C07282=1082.479,167.330,-71.848,174.857,22.621,153.777
C07283=1082.484,167.580,-71.870,174.859,22.623,153.777
C07284=1082.490,167.828,-71.891,174.861,22.624,153.777
C07285=1082.495,168.078,-71.914,174.863,22.627,153.777
C07286=1082.500,168.327,-71.936,174.866,22.629,153.777
C07287=1082.506,168.576,-71.957,174.868,22.631,153.777
C07288=1082.511,168.825,-71.979,174.870,22.633,153.777
C07289=1082.517,169.074,-72.001,174.873,22.635,153.777
C07290=1082.522,169.323,-72.023,174.874,22.637,153.778
C07291=1082.528,169.572,-72.044,174.877,22.639,153.778
C07292=1082.533,169.820,-72.067,174.879,22.641,153.778
C07293=1082.539,170.069,-72.088,174.881,22.643,153.778
C07294=1082.544,170.318,-72.110,174.884,22.645,153.778
C07295=1082.550,170.567,-72.132,174.886,22.647,153.778
C07296=1082.556,170.817,-72.154,174.889,22.649,153.778
C07297=1082.561,171.066,-72.176,174.890,22.651,153.778
C07298=1082.567,171.315,-72.198,174.892,22.653,153.778
C07299=1082.572,171.563,-72.220,174.895,22.655,153.778
C07300=1082.578,171.812,-72.242,174.897,22.657,153.778
C07301=1082.583,172.062,-72.264,174.900,22.659,153.778
C07302=1082.589,172.310,-72.285,174.902,22.661,153.779
C07303=1082.595,172.559,-72.308,174.904,22.663,153.779
C07304=1082.599,172.808,-72.330,174.906,22.665,153.779
C07305=1082.606,173.057,-72.352,174.908,22.667,153.779
C07306=1082.611,173.307,-72.374,174.911,22.669,153.779
C07307=1082.617,173.555,-72.396,174.913,22.671,153.779
C07308=1082.622,173.804,-72.418,174.915,22.673,153.779
C07309=1082.628,174.054,-72.440,174.918,22.675,153.779
C07310=1082.634,174.302,-72.462,174.920,22.677,153.779
C07311=1082.639,174.551,-72.485,174.923,22.679,153.779
C07312=1082.645,174.800,-72.506,174.924,22.681,153.779
C07313=1082.650,175.049,-72.529,174.927,22.683,153.779
C07314=1082.657,175.328,-72.553,174.930,22.685,153.780
C07315=1082.663,175.607,-72.579,174.932,22.688,153.780
C07316=1082.669,175.887,-72.603,174.935,22.689,153.780
C07317=1082.676,176.166,-72.628,174.937,22.692,153.780
C07318=1082.681,176.415,-72.650,174.939,22.693,153.780
C07319=1082.686,176.664,-72.672,174.942,22.696,153.780
C07320=1082.693,176.913,-72.695,174.944,22.697,153.780
C07321=1082.698,177.162,-72.717,174.946,22.700,153.780
C07322=1082.703,177.410,-72.740,174.949,22.702,153.780
C07323=1082.709,177.660,-72.761,174.951,22.704,153.780
C07324=1082.715,177.909,-72.784,174.954,22.706,153.780
C07325=1082.721,178.158,-72.806,174.955,22.708,153.781
C07326=1082.726,178.406,-72.828,174.958,22.709,153.781
C07327=1082.732,178.655,-72.851,174.960,22.711,153.781
C07328=1082.738,178.904,-72.874,174.962,22.713,153.781
C07329=1082.744,179.154,-72.895,174.965,22.715,153.781
C07330=1082.749,179.402,-72.918,174.967,22.717,153.781
C07331=1082.754,179.651,-72.940,174.970,22.719,153.781
C07332=1082.761,179.900,-72.962,174.972,22.722,153.781
C07333=1082.766,180.149,-72.985,174.975,22.723,153.781
C07334=1082.772,180.398,-73.008,174.977,22.725,153.781
C07335=1082.777,180.646,-73.030,174.979,22.727,153.781
C07336=1082.783,180.896,-73.052,174.982,22.729,153.781
C07337=1082.789,181.145,-73.075,174.983,22.730,153.781
C07338=1082.794,181.394,-73.097,174.986,22.733,153.781
C07339=1082.801,181.643,-73.119,174.988,22.735,153.781
C07340=1082.806,181.891,-73.142,174.991,22.737,153.782
C07341=1082.811,182.140,-73.164,174.993,22.739,153.782
C07342=1082.817,182.389,-73.187,174.996,22.740,153.782
C07343=1082.824,182.638,-73.209,174.998,22.743,153.782
C07344=1082.829,182.887,-73.232,175.000,22.744,153.782
C07345=1082.835,183.136,-73.255,175.003,22.746,153.782
C07346=1082.841,183.385,-73.278,175.005,22.749,153.782
C07347=1082.846,183.634,-73.299,175.008,22.750,153.782
C07348=1082.852,183.883,-73.322,175.010,22.752,153.782
C07349=1082.858,184.131,-73.345,175.012,22.754,153.782
C07350=1082.863,184.380,-73.368,175.015,22.756,153.782
C07351=1082.869,184.630,-73.390,175.017,22.758,153.782
C07352=1082.875,184.878,-73.412,175.020,22.760,153.782
C07353=1082.881,185.127,-73.435,175.022,22.762,153.782
C07354=1082.887,185.376,-73.458,175.025,22.764,153.782
C07355=1082.891,185.625,-73.480,175.026,22.766,153.782
C07356=1082.896,185.874,-73.504,175.028,22.768,153.783
C07357=1082.902,186.123,-73.526,175.031,22.770,153.783
C07358=1082.908,186.372,-73.549,175.033,22.772,153.783
C07359=1082.913,186.620,-73.572,175.036,22.774,153.783
C07360=1082.919,186.869,-73.595,175.038,22.776,153.783
C07361=1082.924,187.119,-73.617,175.040,22.778,153.783
C07362=1082.930,187.368,-73.640,175.043,22.780,153.783
C07363=1082.935,187.617,-73.664,175.045,22.782,153.783
C07364=1082.940,187.865,-73.686,175.048,22.784,153.783
C07365=1082.946,188.114,-73.709,175.050,22.786,153.783
C07366=1082.951,188.363,-73.732,175.052,22.788,153.783
C07367=1082.957,188.612,-73.755,175.055,22.791,153.784
C07368=1082.963,188.861,-73.778,175.057,22.792,153.784
C07369=1082.968,189.110,-73.802,175.060,22.795,153.784
C07370=1082.974,189.359,-73.825,175.062,22.796,153.784
C07371=1082.979,189.607,-73.847,175.064,22.799,153.784
C07372=1082.985,189.856,-73.870,175.067,22.800,153.784
C07373=1082.990,190.105,-73.893,175.069,22.803,153.784
C07374=1082.995,190.354,-73.917,175.072,22.804,153.784
C07375=1083.001,190.603,-73.939,175.074,22.807,153.784
C07376=1083.007,190.852,-73.962,175.076,22.809,153.784
C07377=1083.012,191.101,-73.985,175.079,22.811,153.784
C07378=1083.018,191.379,-74.011,175.082,22.814,153.785
C07379=1083.024,191.658,-74.037,175.084,22.815,153.785
C07380=1083.031,191.937,-74.063,175.087,22.818,153.785
C07381=1083.037,192.217,-74.089,175.090,22.820,153.785
C07382=1083.042,192.466,-74.112,175.092,22.822,153.785
C07383=1083.049,192.714,-74.135,175.095,22.824,153.785
C07384=1083.054,192.962,-74.158,175.097,22.826,153.785
C07385=1083.059,193.211,-74.181,175.100,22.828,153.785
C07386=1083.064,193.460,-74.204,175.102,22.830,153.785
C07387=1083.070,193.709,-74.227,175.105,22.832,153.785
C07388=1083.076,193.958,-74.250,175.107,22.834,153.785
C07389=1083.081,194.207,-74.274,175.109,22.836,153.785
C07390=1083.087,194.456,-74.298,175.112,22.838,153.785
C07391=1083.093,194.704,-74.320,175.114,22.840,153.785
C07392=1083.098,194.954,-74.344,175.117,22.842,153.786
C07393=1083.103,195.203,-74.367,175.119,22.844,153.786
C07394=1083.109,195.451,-74.391,175.122,22.846,153.786
C07395=1083.115,195.700,-74.414,175.124,22.848,153.786
C07396=1083.120,195.949,-74.437,175.126,22.850,153.786
C07397=1083.126,196.198,-74.460,175.129,22.852,153.786
C07398=1083.132,196.446,-74.484,175.131,22.854,153.786
C07399=1083.137,196.695,-74.507,175.133,22.856,153.786
C07400=1083.143,196.944,-74.530,175.136,22.858,153.786
C07401=1083.149,197.194,-74.554,175.138,22.860,153.786
C07402=1083.154,197.442,-74.578,175.141,22.862,153.786
C07403=1083.160,197.691,-74.601,175.143,22.864,153.786
C07404=1083.166,197.940,-74.624,175.146,22.867,153.786
C07405=1083.171,198.189,-74.648,175.149,22.868,153.786
C07406=1083.177,198.438,-74.671,175.151,22.870,153.786
C07407=1083.183,198.686,-74.695,175.154,22.872,153.787
C07408=1083.188,198.935,-74.718,175.156,22.874,153.787
C07409=1083.193,199.184,-74.741,175.159,22.876,153.787
C07410=1083.200,199.432,-74.765,175.161,22.878,153.787
C07411=1083.204,199.682,-74.788,175.164,22.880,153.787
C07412=1083.211,199.931,-74.812,175.166,22.882,153.787
C07413=1083.217,200.179,-74.835,175.168,22.884,153.787
C07414=1083.222,200.429,-74.859,175.171,22.886,153.787
C07415=1083.228,200.677,-74.882,175.173,22.888,153.787
C07416=1083.234,200.926,-74.905,175.176,22.890,153.787
C07417=1083.239,201.174,-74.930,175.179,22.892,153.787
C07418=1083.245,201.423,-74.953,175.181,22.894,153.787
C07419=1083.251,201.673,-74.977,175.184,22.896,153.787
C07420=1083.256,201.921,-75.000,175.186,22.898,153.787
C07421=1083.262,202.170,-75.024,175.189,22.900,153.788
C07422=1083.267,202.419,-75.047,175.191,22.902,153.788
C07423=1083.273,202.667,-75.071,175.194,22.904,153.788
C07424=1083.279,202.916,-75.095,175.196,22.906,153.788
C07425=1083.285,203.165,-75.119,175.199,22.908,153.788
C07426=1083.290,203.414,-75.143,175.201,22.910,153.788
C07427=1083.295,203.663,-75.166,175.204,22.912,153.788
C07428=1083.301,203.911,-75.190,175.207,22.914,153.788
C07429=1083.307,204.160,-75.214,175.209,22.916,153.788
C07430=1083.312,204.409,-75.237,175.211,22.918,153.788
C07431=1083.318,204.658,-75.261,175.214,22.920,153.788
C07432=1083.323,204.907,-75.285,175.216,22.923,153.788
C07433=1083.329,205.156,-75.309,175.219,22.924,153.788
C07434=1083.335,205.404,-75.333,175.221,22.927,153.789
C07435=1083.340,205.653,-75.358,175.224,22.928,153.789
C07436=1083.346,205.902,-75.380,175.227,22.931,153.789
C07437=1083.351,206.150,-75.405,175.229,22.933,153.789
C07438=1083.357,206.400,-75.429,175.232,22.935,153.789
C07439=1083.363,206.649,-75.452,175.234,22.937,153.789
C07440=1083.368,206.897,-75.477,175.237,22.939,153.789
C07441=1083.373,207.146,-75.501,175.239,22.941,153.789
C07442=1083.397,208.176,-75.600,175.328,22.988,153.786
C07443=1083.406,208.569,-75.639,175.332,22.993,153.787
C07444=1083.415,208.961,-75.677,175.336,22.997,153.787
C07445=1083.423,209.353,-75.716,175.340,23.002,153.788
C07446=1083.432,209.746,-75.754,175.344,23.007,153.788
C07447=1083.438,209.995,-75.779,175.346,23.010,153.789
C07448=1083.444,210.243,-75.804,175.349,23.013,153.789
C07449=1083.450,210.492,-75.828,175.351,23.016,153.789
C07450=1083.455,210.741,-75.853,175.353,23.019,153.789
C07451=1083.460,210.990,-75.877,175.356,23.022,153.790
C07452=1083.466,211.238,-75.902,175.358,23.025,153.790
C07453=1083.472,211.487,-75.927,175.360,23.027,153.790
C07454=1083.478,211.736,-75.951,175.363,23.031,153.791
C07455=1083.483,211.984,-75.976,175.365,23.034,153.791
C07456=1083.489,212.233,-76.001,175.368,23.037,153.791
C07457=1083.494,212.482,-76.025,175.371,23.040,153.791
C07458=1083.501,212.731,-76.050,175.373,23.043,153.792
C07459=1083.506,212.979,-76.075,175.375,23.045,153.792
C07460=1083.512,213.229,-76.099,175.378,23.049,153.792
C07461=1083.517,213.476,-76.124,175.380,23.051,153.793
C07462=1083.523,213.726,-76.149,175.382,23.055,153.793
C07463=1083.528,213.975,-76.174,175.385,23.058,153.793
C07464=1083.534,214.223,-76.199,175.387,23.061,153.793
C07465=1083.539,214.472,-76.223,175.389,23.063,153.794
C07466=1083.546,214.721,-76.249,175.392,23.067,153.794
C07467=1083.551,214.969,-76.273,175.394,23.070,153.794
C07468=1083.557,215.218,-76.298,175.397,23.073,153.795
C07469=1083.562,215.467,-76.323,175.400,23.076,153.795
C07470=1083.568,215.715,-76.348,175.402,23.079,153.795
C07471=1083.573,215.964,-76.373,175.405,23.082,153.796
C07472=1083.579,216.213,-76.398,175.407,23.085,153.796
C07473=1083.585,216.461,-76.422,175.409,23.088,153.796
C07474=1083.590,216.710,-76.448,175.412,23.091,153.796
C07475=1083.596,216.959,-76.472,175.414,23.094,153.797
C07476=1083.602,217.208,-76.498,175.417,23.097,153.797
C07477=1083.607,217.456,-76.522,175.419,23.100,153.797
C07478=1083.612,217.705,-76.548,175.421,23.103,153.798
C07479=1083.619,217.954,-76.573,175.425,23.106,153.798
C07480=1083.624,218.202,-76.598,175.427,23.108,153.798
C07481=1083.630,218.451,-76.623,175.429,23.112,153.799
C07482=1083.636,218.699,-76.648,175.432,23.115,153.799
C07483=1083.641,218.949,-76.673,175.434,23.118,153.799
C07484=1083.647,219.197,-76.698,175.437,23.121,153.799
C07485=1083.653,219.445,-76.723,175.439,23.124,153.800
C07486=1083.658,219.695,-76.749,175.441,23.126,153.800
C07487=1083.664,219.943,-76.774,175.444,23.130,153.800
C07488=1083.670,220.191,-76.799,175.446,23.132,153.800
C07489=1083.676,220.441,-76.824,175.449,23.136,153.801
C07490=1083.681,220.689,-76.849,175.451,23.139,153.801
C07491=1083.687,220.938,-76.874,175.454,23.142,153.801
C07492=1083.693,221.186,-76.900,175.457,23.145,153.802
C07493=1083.697,221.435,-76.925,175.459,23.148,153.802
C07494=1083.704,221.684,-76.950,175.462,23.151,153.802
C07495=1083.713,222.080,-76.990,175.465,23.155,153.803
C07496=1083.722,222.477,-77.031,175.470,23.160,153.803
C07497=1083.730,222.873,-77.072,175.474,23.165,153.804
C07498=1083.740,223.270,-77.112,175.477,23.170,153.804
C07499=1083.745,223.518,-77.138,175.480,23.173,153.804
C07500=1083.751,223.767,-77.163,175.482,23.176,153.805
C07501=1083.757,224.016,-77.189,175.485,23.179,153.805
C07502=1083.762,224.264,-77.213,175.487,23.182,153.805
C07503=1083.768,224.513,-77.239,175.491,23.185,153.806
C07504=1083.774,224.762,-77.264,175.493,23.188,153.806
C07505=1083.779,225.010,-77.290,175.495,23.191,153.806
C07506=1083.785,225.259,-77.315,175.498,23.194,153.807
C07507=1083.790,225.508,-77.341,175.500,23.197,153.807
C07508=1083.797,225.757,-77.366,175.503,23.200,153.807
C07509=1083.801,226.005,-77.392,175.505,23.203,153.807
C07510=1083.807,226.254,-77.418,175.508,23.206,153.808
C07511=1083.813,226.502,-77.443,175.510,23.209,153.808
C07512=1083.819,226.751,-77.469,175.512,23.212,153.808
C07513=1083.824,226.999,-77.494,175.515,23.215,153.809
C07514=1083.830,227.248,-77.520,175.518,23.218,153.809
C07515=1083.836,227.496,-77.546,175.521,23.221,153.809
C07516=1083.842,227.745,-77.572,175.523,23.224,153.809
C07517=1083.847,227.993,-77.597,175.526,23.227,153.810
C07518=1083.853,228.242,-77.623,175.528,23.230,153.810
C07519=1083.858,228.491,-77.649,175.530,23.233,153.810
C07520=1083.864,228.740,-77.674,175.533,23.236,153.811
C07521=1083.870,228.989,-77.700,175.535,23.239,153.811
C07522=1083.875,229.237,-77.725,175.538,23.242,153.811
C07523=1083.881,229.485,-77.752,175.540,23.245,153.812
C07524=1083.887,229.734,-77.778,175.543,23.248,153.812
C07525=1083.893,229.983,-77.803,175.546,23.251,153.812
C07526=1083.898,230.232,-77.829,175.549,23.254,153.812
C07527=1083.904,230.480,-77.856,175.551,23.257,153.813
C07528=1083.910,230.728,-77.881,175.554,23.260,153.813
C07529=1083.915,230.977,-77.907,175.556,23.264,153.813
C07530=1083.921,231.226,-77.933,175.559,23.267,153.814
C07531=1083.926,231.475,-77.959,175.561,23.269,153.814
C07532=1083.933,231.723,-77.985,175.563,23.272,153.814
C07533=1083.938,231.972,-78.010,175.566,23.275,153.814
C07534=1083.943,232.220,-78.037,175.568,23.279,153.815
C07535=1083.949,232.469,-78.063,175.571,23.282,153.815
C07536=1083.955,232.718,-78.088,175.574,23.285,153.815
C07537=1083.961,232.966,-78.115,175.577,23.288,153.816
C07538=1083.966,233.215,-78.141,175.579,23.291,153.816
C07539=1083.972,233.464,-78.167,175.582,23.294,153.816
C07540=1083.977,233.712,-78.193,175.584,23.297,153.817
C07541=1083.983,233.961,-78.219,175.587,23.300,153.817
C07542=1083.989,234.209,-78.245,175.589,23.303,153.817
C07543=1083.994,234.458,-78.271,175.592,23.306,153.817
C07544=1084.000,234.706,-78.297,175.594,23.309,153.818
C07545=1084.005,234.955,-78.323,175.597,23.312,153.818
C07546=1084.011,235.204,-78.349,175.599,23.315,153.818
C07547=1084.020,235.591,-78.390,175.604,23.320,153.819
C07548=1084.029,235.979,-78.432,175.608,23.325,153.819
C07549=1084.037,236.367,-78.472,175.612,23.330,153.820
C07550=1084.047,236.755,-78.513,175.616,23.334,153.820
C07551=1084.052,237.004,-78.539,175.619,23.338,153.821
C07552=1084.058,237.253,-78.566,175.621,23.340,153.821
C07553=1084.063,237.500,-78.592,175.624,23.344,153.821
C07554=1084.069,237.749,-78.618,175.626,23.347,153.821
C07555=1084.075,237.998,-78.645,175.629,23.350,153.822
C07556=1084.080,238.247,-78.671,175.631,23.353,153.822
C07557=1084.086,238.495,-78.697,175.634,23.356,153.822
C07558=1084.092,238.743,-78.724,175.637,23.359,153.823
C07559=1084.097,238.992,-78.750,175.639,23.362,153.823
C07560=1084.103,239.241,-78.777,175.642,23.365,153.823
C07561=1084.109,239.489,-78.803,175.645,23.368,153.824
C07562=1084.114,239.737,-78.830,175.647,23.371,153.824
C07563=1084.120,239.986,-78.856,175.650,23.374,153.824
C07564=1084.126,240.235,-78.883,175.652,23.377,153.825
C07565=1084.132,240.484,-78.910,175.655,23.380,153.825
C07566=1084.138,240.732,-78.936,175.657,23.383,153.825
C07567=1084.143,240.981,-78.962,175.660,23.386,153.825
C07568=1084.149,241.230,-78.989,175.662,23.389,153.826
C07569=1084.155,241.478,-79.015,175.666,23.392,153.826
C07570=1084.160,241.727,-79.043,175.668,23.395,153.826
C07571=1084.166,241.975,-79.069,175.671,23.399,153.827
C07572=1084.171,242.224,-79.095,175.674,23.402,153.827
C07573=1084.177,242.472,-79.122,175.676,23.405,153.827
C07574=1084.183,242.721,-79.149,175.679,23.408,153.827
C07575=1084.188,242.969,-79.175,175.681,23.410,153.828
C07576=1084.194,243.217,-79.202,175.684,23.414,153.828
C07577=1084.200,243.466,-79.229,175.686,23.417,153.828
C07578=1084.205,243.714,-79.256,175.689,23.420,153.829
C07579=1084.211,243.963,-79.282,175.691,23.423,153.829
C07580=1084.217,244.212,-79.309,175.694,23.426,153.829
C07581=1084.223,244.460,-79.336,175.697,23.429,153.830
C07582=1084.228,244.709,-79.363,175.700,23.432,153.830
C07583=1084.234,244.957,-79.390,175.703,23.436,153.830
C07584=1084.239,245.206,-79.417,175.705,23.439,153.831
C07585=1084.244,245.454,-79.444,175.708,23.442,153.831
C07586=1084.250,245.703,-79.471,175.710,23.445,153.831
C07587=1084.256,245.951,-79.497,175.713,23.448,153.832
C07588=1084.262,246.199,-79.524,175.715,23.451,153.832
C07589=1084.267,246.449,-79.551,175.718,23.454,153.832
C07590=1084.273,246.697,-79.578,175.721,23.457,153.832
C07591=1084.279,246.945,-79.605,175.723,23.460,153.833
C07592=1084.284,247.194,-79.632,175.726,23.464,153.833
C07593=1084.290,247.442,-79.659,175.729,23.466,153.833
C07594=1084.295,247.690,-79.687,175.731,23.470,153.834
C07595=1084.301,247.939,-79.713,175.734,23.473,153.834
C07596=1084.307,248.187,-79.740,175.737,23.476,153.834
C07597=1084.312,248.437,-79.768,175.740,23.480,153.835
C07598=1084.318,248.685,-79.794,175.742,23.482,153.835
C07599=1084.326,249.066,-79.835,175.746,23.487,153.835
C07600=1084.335,249.447,-79.878,175.750,23.492,153.836
C07601=1084.343,249.828,-79.920,175.755,23.497,153.836
C07602=1084.351,250.209,-79.961,175.758,23.502,153.837
C07603=1084.357,250.457,-79.988,175.761,23.505,153.837
C07604=1084.363,250.706,-80.016,175.763,23.508,153.838
C07605=1084.369,250.955,-80.043,175.766,23.511,153.838
C07606=1084.374,251.203,-80.071,175.769,23.515,153.838
C07607=1084.380,251.451,-80.097,175.771,23.517,153.838
C07608=1084.385,251.700,-80.124,175.774,23.521,153.839
C07609=1084.392,251.948,-80.152,175.777,23.524,153.839
C07610=1084.397,252.197,-80.179,175.780,23.527,153.839
C07611=1084.402,252.445,-80.207,175.783,23.530,153.840
C07612=1084.408,252.693,-80.234,175.785,23.533,153.840
C07613=1084.413,252.943,-80.262,175.788,23.536,153.840
C07614=1084.419,253.190,-80.289,175.790,23.540,153.841
C07615=1084.424,253.439,-80.316,175.793,23.543,153.841
C07616=1084.431,253.687,-80.344,175.796,23.546,153.841
C07617=1084.436,253.936,-80.371,175.798,23.549,153.842
C07618=1084.442,254.184,-80.399,175.801,23.552,153.842
C07619=1084.447,254.433,-80.426,175.803,23.555,153.842
C07620=1084.453,254.681,-80.454,175.806,23.559,153.843
C07621=1084.459,254.930,-80.481,175.809,23.562,153.843
C07622=1084.464,255.178,-80.509,175.812,23.564,153.843
C07623=1084.470,255.427,-80.536,175.815,23.568,153.844
C07624=1084.476,255.675,-80.564,175.818,23.571,153.844
C07625=1084.481,255.923,-80.592,175.820,23.574,153.844
C07626=1084.488,256.172,-80.619,175.823,23.577,153.845
C07627=1084.493,256.420,-80.647,175.825,23.580,153.845
C07628=1084.498,256.669,-80.674,175.828,23.583,153.845
C07629=1084.505,256.917,-80.702,175.831,23.587,153.845
C07630=1084.510,257.165,-80.730,175.833,23.590,153.846
C07631=1084.515,257.414,-80.757,175.836,23.593,153.846
C07632=1084.522,257.662,-80.785,175.839,23.596,153.846
C07633=1084.527,257.910,-80.812,175.841,23.599,153.847
C07634=1084.533,258.158,-80.840,175.844,23.602,153.847
C07635=1084.539,258.408,-80.867,175.848,23.606,153.847
C07636=1084.544,258.656,-80.895,175.850,23.608,153.848
C07637=1084.550,258.904,-80.924,175.853,23.612,153.848
C07638=1084.556,259.152,-80.951,175.856,23.615,153.848
C07639=1084.562,259.401,-80.979,175.858,23.618,153.849
C07640=1084.567,259.650,-81.007,175.861,23.621,153.849
C07641=1084.573,259.897,-81.034,175.863,23.624,153.849
C07642=1084.579,260.146,-81.062,175.866,23.627,153.850
C07643=1084.585,260.394,-81.090,175.869,23.630,153.850
C07644=1084.590,260.643,-81.118,175.871,23.634,153.850
C07645=1084.596,260.891,-81.145,175.874,23.637,153.851
C07646=1084.602,261.140,-81.174,175.878,23.640,153.851
C07647=1084.608,261.388,-81.202,175.880,23.643,153.851
C07648=1084.614,261.637,-81.230,175.883,23.646,153.852
C07649=1084.620,261.884,-81.257,175.886,23.649,153.852
C07650=1084.626,262.133,-81.286,175.888,23.652,153.852
C07651=1084.635,262.511,-81.328,175.892,23.657,153.853
C07652=1084.644,262.889,-81.371,175.897,23.662,153.853
C07653=1084.652,263.268,-81.413,175.901,23.667,153.854
C07654=1084.661,263.647,-81.456,175.905,23.671,153.854
C07655=1084.666,263.895,-81.484,175.908,23.675,153.854
C07656=1084.672,264.144,-81.512,175.910,23.678,153.855
C07657=1084.678,264.391,-81.540,175.914,23.681,153.855
C07658=1084.685,264.639,-81.569,175.916,23.685,153.855
C07659=1084.690,264.888,-81.597,175.919,23.687,153.856
C07660=1084.695,265.137,-81.625,175.922,23.691,153.856
C07661=1084.701,265.385,-81.653,175.925,23.694,153.856
C07662=1084.707,265.633,-81.682,175.927,23.697,153.857
C07663=1084.712,265.881,-81.710,175.930,23.700,153.857
C07664=1084.718,266.130,-81.738,175.933,23.703,153.857
C07665=1084.723,266.378,-81.766,175.935,23.707,153.858
C07666=1084.729,266.626,-81.795,175.938,23.710,153.858
C07667=1084.735,266.874,-81.823,175.941,23.713,153.858
C07668=1084.741,267.123,-81.851,175.944,23.717,153.859
C07669=1084.747,267.372,-81.880,175.946,23.720,153.859
C07670=1084.752,267.620,-81.908,175.949,23.723,153.859
C07671=1084.758,267.868,-81.937,175.952,23.726,153.860
C07672=1084.764,268.116,-81.965,175.954,23.729,153.860
C07673=1084.770,268.365,-81.993,175.958,23.732,153.860
C07674=1084.775,268.612,-82.022,175.960,23.736,153.861
C07675=1084.781,268.861,-82.050,175.964,23.739,153.861
C07676=1084.787,269.110,-82.078,175.966,23.742,153.861
C07677=1084.792,269.358,-82.108,175.969,23.745,153.862
C07678=1084.798,269.606,-82.136,175.972,23.749,153.862
C07679=1084.803,269.854,-82.164,175.974,23.752,153.862
C07680=1084.810,270.103,-82.193,175.977,23.755,153.863
C07681=1084.815,270.351,-82.221,175.980,23.758,153.863
C07682=1084.821,270.599,-82.249,175.983,23.762,153.863
C07683=1084.826,270.848,-82.279,175.985,23.765,153.864
C07684=1084.832,271.097,-82.307,175.988,23.768,153.864
C07685=1084.838,271.344,-82.336,175.991,23.772,153.864
C07686=1084.844,271.593,-82.364,175.993,23.775,153.865
C07687=1084.849,271.841,-82.394,175.996,23.778,153.865
C07688=1084.855,272.089,-82.422,175.999,23.781,153.866
C07689=1084.861,272.337,-82.451,176.002,23.785,153.866
C07690=1084.866,272.585,-82.479,176.004,23.788,153.866
C07691=1084.872,272.834,-82.508,176.008,23.791,153.867
C07692=1084.878,273.083,-82.537,176.010,23.795,153.867
C07693=1084.884,273.331,-82.566,176.014,23.798,153.867
C07694=1084.889,273.579,-82.594,176.016,23.801,153.868
C07695=1084.895,273.827,-82.623,176.019,23.804,153.868
C07696=1084.901,274.075,-82.652,176.022,23.808,153.868
C07697=1084.906,274.323,-82.680,176.025,23.811,153.869
C07698=1084.912,274.572,-82.710,176.027,23.814,153.869
C07699=1084.918,274.820,-82.739,176.030,23.818,153.869
C07700=1084.924,275.068,-82.767,176.033,23.821,153.870
C07701=1084.929,275.316,-82.797,176.036,23.824,153.870
C07702=1084.935,275.565,-82.826,176.038,23.827,153.870
C07703=1084.944,275.946,-82.870,176.043,23.832,153.871
C07704=1084.953,276.328,-82.914,176.047,23.837,153.871
C07705=1084.961,276.708,-82.959,176.052,23.843,153.872
C07706=1084.970,277.089,-83.003,176.056,23.848,153.873
C07707=1084.976,277.338,-83.033,176.058,23.851,153.873
C07708=1084.981,277.586,-83.062,176.061,23.854,153.873
C07709=1084.988,277.834,-83.091,176.064,23.857,153.874
C07710=1084.992,278.082,-83.120,176.067,23.861,153.874
C07711=1084.998,278.331,-83.149,176.069,23.864,153.874
C07712=1085.004,278.579,-83.178,176.072,23.867,153.875
C07713=1085.010,278.827,-83.207,176.075,23.871,153.875
C07714=1085.016,279.076,-83.237,176.078,23.874,153.875
C07715=1085.021,279.323,-83.266,176.081,23.878,153.876
C07716=1085.027,279.571,-83.295,176.084,23.881,153.876
C07717=1085.033,279.820,-83.324,176.087,23.884,153.877
C07718=1085.039,280.068,-83.354,176.090,23.888,153.877
C07719=1085.045,280.316,-83.383,176.093,23.891,153.877
C07720=1085.050,280.565,-83.413,176.096,23.894,153.878
C07721=1085.056,280.812,-83.441,176.098,23.898,153.878
C07722=1085.061,281.060,-83.471,176.101,23.901,153.878
C07723=1085.068,281.309,-83.500,176.104,23.904,153.879
C07724=1085.073,281.557,-83.530,176.107,23.908,153.879
C07725=1085.079,281.805,-83.559,176.110,23.911,153.880
C07726=1085.084,282.054,-83.589,176.112,23.915,153.880
C07727=1085.090,282.301,-83.618,176.115,23.918,153.880
C07728=1085.095,282.550,-83.647,176.118,23.921,153.881
C07729=1085.101,282.798,-83.677,176.121,23.925,153.881
C07730=1085.107,283.046,-83.706,176.124,23.928,153.881
C07731=1085.113,283.295,-83.736,176.126,23.931,153.882
C07732=1085.119,283.543,-83.766,176.129,23.935,153.882
C07733=1085.123,283.790,-83.795,176.132,23.938,153.883
C07734=1085.130,284.039,-83.824,176.135,23.942,153.883
C07735=1085.135,284.287,-83.854,176.138,23.945,153.883
C07736=1085.141,284.535,-83.884,176.141,23.949,153.884
C07737=1085.147,284.783,-83.913,176.143,23.952,153.884
C07738=1085.153,285.031,-83.943,176.146,23.955,153.885
C07739=1085.158,285.280,-83.973,176.149,23.959,153.885
C07740=1085.164,285.528,-84.002,176.152,23.962,153.885
C07741=1085.170,285.776,-84.033,176.155,23.966,153.886
C07742=1085.176,286.024,-84.062,176.158,23.969,153.886
C07743=1085.181,286.273,-84.091,176.160,23.972,153.886
C07744=1085.187,286.520,-84.122,176.163,23.976,153.887
C07745=1085.193,286.769,-84.151,176.166,23.979,153.887
C07746=1085.199,287.017,-84.180,176.169,23.983,153.888
C07747=1085.205,287.265,-84.211,176.172,23.986,153.888
C07748=1085.210,287.513,-84.240,176.175,23.989,153.888
C07749=1085.215,287.760,-84.270,176.177,23.993,153.889
C07750=1085.221,288.009,-84.300,176.180,23.996,153.889
C07751=1085.227,288.257,-84.329,176.183,24.000,153.889
C07752=1085.233,288.505,-84.359,176.186,24.003,153.890
C07753=1085.239,288.754,-84.389,176.189,24.006,153.890
C07754=1085.245,289.002,-84.420,176.192,24.010,153.891
C07755=1085.253,289.392,-84.466,176.197,24.015,153.891
C07756=1085.263,289.783,-84.513,176.201,24.021,153.892
C07757=1085.272,290.174,-84.561,176.206,24.026,153.892
C07758=1085.281,290.565,-84.608,176.210,24.032,153.893
C07759=1085.287,290.813,-84.638,176.213,24.035,153.893
C07760=1085.292,291.061,-84.668,176.216,24.039,153.894
C07761=1085.298,291.309,-84.698,176.219,24.042,153.894
C07762=1085.304,291.557,-84.729,176.222,24.046,153.895
C07763=1085.309,291.805,-84.758,176.225,24.049,153.895
C07764=1085.315,292.053,-84.789,176.227,24.053,153.895
C07765=1085.321,292.301,-84.819,176.230,24.056,153.896
C07766=1085.326,292.549,-84.849,176.233,24.060,153.896
C07767=1085.333,292.798,-84.879,176.236,24.063,153.897
C07768=1085.339,293.046,-84.910,176.239,24.067,153.897
C07769=1085.344,293.294,-84.939,176.242,24.071,153.897
C07770=1085.350,293.542,-84.970,176.245,24.074,153.898
C07771=1085.355,293.790,-85.001,176.248,24.078,153.898
C07772=1085.361,294.038,-85.031,176.251,24.081,153.899
C07773=1085.367,294.286,-85.061,176.253,24.084,153.899
C07774=1085.372,294.534,-85.091,176.256,24.088,153.900
C07775=1085.378,294.782,-85.121,176.259,24.092,153.900
C07776=1085.384,295.030,-85.152,176.262,24.095,153.900
C07777=1085.390,295.278,-85.182,176.265,24.099,153.901
C07778=1085.396,295.526,-85.213,176.268,24.102,153.901
C07779=1085.402,295.774,-85.243,176.271,24.106,153.902
C07780=1085.407,296.022,-85.274,176.274,24.109,153.902
C07781=1085.413,296.270,-85.304,176.277,24.113,153.902
C07782=1085.418,296.518,-85.334,176.280,24.117,153.903
C07783=1085.425,296.767,-85.365,176.283,24.120,153.903
C07784=1085.431,297.015,-85.395,176.286,24.124,153.904
C07785=1085.436,297.263,-85.426,176.288,24.127,153.904
C07786=1085.441,297.511,-85.456,176.291,24.130,153.905
C07787=1085.447,297.758,-85.487,176.294,24.134,153.905
C07788=1085.453,298.006,-85.517,176.297,24.138,153.905
C07789=1085.459,298.255,-85.548,176.300,24.141,153.906
C07790=1085.465,298.503,-85.579,176.303,24.145,153.906
C07791=1085.470,298.750,-85.610,176.306,24.149,153.907
C07792=1085.476,298.998,-85.641,176.309,24.152,153.907
C07793=1085.482,299.246,-85.671,176.312,24.156,153.908
C07794=1085.487,299.494,-85.702,176.315,24.160,153.908
C07795=1085.493,299.742,-85.732,176.318,24.164,153.908
C07796=1085.498,299.991,-85.764,176.321,24.167,153.909
C07797=1085.504,300.239,-85.794,176.324,24.171,153.909
C07798=1085.509,300.487,-85.825,176.326,24.175,153.910
C07799=1085.515,300.734,-85.856,176.329,24.178,153.910
C07800=1085.520,300.982,-85.887,176.332,24.182,153.911
C07801=1085.527,301.231,-85.918,176.335,24.185,153.911
C07802=1085.532,301.479,-85.949,176.338,24.190,153.912
C07803=1085.538,301.726,-85.980,176.341,24.193,153.912
C07804=1085.543,301.974,-86.011,176.343,24.196,153.912
C07805=1085.549,302.222,-86.041,176.346,24.200,153.913
C07806=1085.555,302.471,-86.072,176.349,24.204,153.913
C07807=1085.564,302.875,-86.123,176.354,24.210,153.914
C07808=1085.573,303.280,-86.173,176.359,24.216,153.915
C07809=1085.583,303.685,-86.224,176.364,24.222,153.916
C07810=1085.592,304.089,-86.275,176.368,24.228,153.916
C07811=1085.597,304.338,-86.306,176.371,24.232,153.917
C07812=1085.604,304.586,-86.337,176.374,24.236,153.917
C07813=1085.609,304.834,-86.369,176.377,24.239,153.918
C07814=1085.615,305.081,-86.399,176.380,24.243,153.918
C07815=1085.621,305.330,-86.431,176.383,24.247,153.919
C07816=1085.627,305.577,-86.461,176.386,24.250,153.919
C07817=1085.632,305.825,-86.493,176.389,24.254,153.919
C07818=1085.638,306.074,-86.524,176.392,24.258,153.920
C07819=1085.644,306.321,-86.555,176.395,24.261,153.920
C07820=1085.649,306.569,-86.586,176.398,24.265,153.921
C07821=1085.656,306.817,-86.618,176.401,24.269,153.921
C07822=1085.661,307.064,-86.649,176.405,24.273,153.922
C07823=1085.667,307.313,-86.681,176.407,24.277,153.922
C07824=1085.673,307.561,-86.712,176.410,24.281,153.923
C07825=1085.678,307.809,-86.743,176.413,24.284,153.923
C07826=1085.684,308.057,-86.775,176.416,24.288,153.924
C07827=1085.690,308.304,-86.806,176.419,24.292,153.924
C07828=1085.696,308.553,-86.837,176.422,24.295,153.925
C07829=1085.702,308.800,-86.868,176.425,24.299,153.925
C07830=1085.708,309.048,-86.900,176.428,24.303,153.925
C07831=1085.713,309.296,-86.931,176.431,24.307,153.926
C07832=1085.720,309.544,-86.963,176.434,24.310,153.926
C07833=1085.725,309.792,-86.994,176.437,24.315,153.927
C07834=1085.731,310.040,-87.026,176.440,24.318,153.927
C07835=1085.737,310.288,-87.057,176.443,24.322,153.928
C07836=1085.743,310.536,-87.089,176.446,24.326,153.928
C07837=1085.748,310.784,-87.120,176.449,24.329,153.929
C07838=1085.754,311.032,-87.152,176.452,24.333,153.929
C07839=1085.760,311.279,-87.183,176.455,24.337,153.930
C07840=1085.766,311.528,-87.215,176.457,24.341,153.930
C07841=1085.771,311.775,-87.246,176.460,24.344,153.931
C07842=1085.778,312.023,-87.278,176.463,24.348,153.931
C07843=1085.783,312.271,-87.309,176.466,24.352,153.932
C07844=1085.789,312.519,-87.341,176.469,24.355,153.932
C07845=1085.795,312.767,-87.373,176.472,24.360,153.933
C07846=1085.802,313.014,-87.405,176.475,24.363,153.933
C07847=1085.807,313.263,-87.437,176.478,24.367,153.934
C07848=1085.813,313.510,-87.468,176.481,24.371,153.934
C07849=1085.819,313.758,-87.500,176.485,24.375,153.934
C07850=1085.826,314.006,-87.532,176.488,24.379,153.935
C07851=1085.831,314.254,-87.563,176.491,24.383,153.935
C07852=1085.837,314.502,-87.595,176.494,24.386,153.936
C07853=1085.843,314.750,-87.627,176.497,24.390,153.936
C07854=1085.848,314.998,-87.659,176.500,24.394,153.937
C07855=1085.854,315.246,-87.691,176.502,24.398,153.937
C07856=1085.860,315.493,-87.723,176.505,24.402,153.938
C07857=1085.866,315.742,-87.755,176.508,24.406,153.938
C07858=1085.872,315.990,-87.787,176.511,24.410,153.939
C07859=1085.880,316.398,-87.840,176.516,24.417,153.940
C07860=1085.890,316.805,-87.893,176.521,24.423,153.941
C07861=1085.899,317.213,-87.945,176.526,24.429,153.942
C07862=1085.909,317.621,-87.998,176.531,24.436,153.942
C07863=1085.914,317.869,-88.030,176.534,24.440,153.943
C07864=1085.920,318.117,-88.063,176.536,24.444,153.944
C07865=1085.925,318.364,-88.095,176.539,24.448,153.944
C07866=1085.931,318.612,-88.127,176.542,24.452,153.945
C07867=1085.937,318.859,-88.159,176.546,24.457,153.945
C07868=1085.942,319.108,-88.192,176.549,24.461,153.946
C07869=1085.948,319.356,-88.224,176.552,24.464,153.946
C07870=1085.954,319.603,-88.256,176.555,24.468,153.947
C07871=1085.960,319.851,-88.288,176.558,24.472,153.947
C07872=1085.965,320.100,-88.321,176.560,24.476,153.948
C07873=1085.971,320.346,-88.353,176.563,24.480,153.948
C07874=1085.977,320.595,-88.385,176.566,24.484,153.949
C07875=1085.983,320.843,-88.417,176.569,24.488,153.949
C07876=1085.989,321.091,-88.451,176.573,24.493,153.950
C07877=1085.994,321.338,-88.482,176.576,24.497,153.950
C07878=1086.000,321.586,-88.515,176.579,24.501,153.951
C07879=1086.006,321.834,-88.547,176.581,24.505,153.952
C07880=1086.012,322.082,-88.580,176.584,24.509,153.952
C07881=1086.017,322.330,-88.612,176.587,24.513,153.953
C07882=1086.023,322.577,-88.645,176.590,24.517,153.953
C07883=1086.029,322.826,-88.677,176.593,24.521,153.954
C07884=1086.035,323.073,-88.710,176.597,24.525,153.954
C07885=1086.041,323.321,-88.743,176.600,24.529,153.955
C07886=1086.046,323.569,-88.775,176.602,24.534,153.956
C07887=1086.052,323.816,-88.808,176.605,24.538,153.956
C07888=1086.058,324.065,-88.840,176.608,24.542,153.957
C07889=1086.064,324.312,-88.873,176.611,24.546,153.957
C07890=1086.070,324.560,-88.906,176.615,24.550,153.958
C07891=1086.076,324.808,-88.938,176.618,24.554,153.958
C07892=1086.081,325.055,-88.971,176.621,24.558,153.959
C07893=1086.087,325.303,-89.004,176.623,24.562,153.959
C07894=1086.093,325.551,-89.036,176.626,24.566,153.960
C07895=1086.099,325.799,-89.069,176.629,24.570,153.960
C07896=1086.105,326.047,-89.102,176.633,24.575,153.961
C07897=1086.111,326.294,-89.134,176.636,24.579,153.962
C07898=1086.117,326.543,-89.167,176.639,24.583,153.962
C07899=1086.123,326.790,-89.200,176.642,24.587,153.963
C07900=1086.129,327.038,-89.233,176.644,24.591,153.963
C07901=1086.135,327.286,-89.266,176.647,24.595,153.964
C07902=1086.141,327.533,-89.298,176.651,24.600,153.964
C07903=1086.146,327.781,-89.332,176.654,24.604,153.965
C07904=1086.152,328.029,-89.364,176.657,24.608,153.966
C07905=1086.158,328.277,-89.397,176.660,24.612,153.966
C07906=1086.164,328.524,-89.430,176.662,24.616,153.967
C07907=1086.169,328.772,-89.463,176.666,24.621,153.967
C07908=1086.176,329.020,-89.496,176.669,24.625,153.968
C07909=1086.182,329.268,-89.529,176.672,24.629,153.968
C07910=1086.188,329.515,-89.562,176.675,24.633,153.969
C07911=1086.198,329.916,-89.616,176.680,24.640,153.970
C07912=1086.207,330.318,-89.669,176.685,24.646,153.971
C07913=1086.217,330.719,-89.723,176.690,24.654,153.972
C07914=1086.227,331.120,-89.776,176.695,24.661,153.973
C07915=1086.233,331.367,-89.810,176.698,24.665,153.973
C07916=1086.239,331.615,-89.843,176.701,24.669,153.974
C07917=1086.244,331.863,-89.876,176.704,24.673,153.975
C07918=1086.251,332.111,-89.909,176.707,24.678,153.975
C07919=1086.256,332.358,-89.942,176.710,24.682,153.976
C07920=1086.262,332.606,-89.975,176.713,24.686,153.976
C07921=1086.268,332.854,-90.009,176.716,24.690,153.977
C07922=1086.274,333.101,-90.042,176.720,24.695,153.978
C07923=1086.279,333.349,-90.075,176.722,24.699,153.978
C07924=1086.285,333.597,-90.109,176.725,24.704,153.979
C07925=1086.291,333.845,-90.142,176.728,24.708,153.979
C07926=1086.296,334.092,-90.176,176.732,24.713,153.980
C07927=1086.303,334.340,-90.209,176.735,24.717,153.981
C07928=1086.308,334.588,-90.242,176.737,24.721,153.981
C07929=1086.314,334.835,-90.276,176.740,24.726,153.982
C07930=1086.320,335.083,-90.310,176.744,24.730,153.983
C07931=1086.326,335.332,-90.343,176.747,24.734,153.983
C07932=1086.332,335.579,-90.377,176.750,24.739,153.984
C07933=1086.338,335.826,-90.410,176.753,24.744,153.985
C07934=1086.344,336.074,-90.444,176.756,24.748,153.985
C07935=1086.349,336.322,-90.478,176.759,24.752,153.986
C07936=1086.355,336.570,-90.511,176.762,24.757,153.987
C07937=1086.361,336.817,-90.545,176.765,24.761,153.987
C07938=1086.368,337.065,-90.578,176.768,24.765,153.988
C07939=1086.374,337.312,-90.612,176.771,24.770,153.988
C07940=1086.379,337.560,-90.645,176.775,24.775,153.989
C07941=1086.385,337.808,-90.679,176.777,24.779,153.990
C07942=1086.391,338.055,-90.713,176.780,24.784,153.990
C07943=1086.396,338.303,-90.747,176.784,24.788,153.991
C07944=1086.403,338.551,-90.781,176.787,24.792,153.992
C07945=1086.408,338.799,-90.815,176.790,24.797,153.992
C07946=1086.414,339.046,-90.849,176.793,24.802,153.993
C07947=1086.420,339.294,-90.882,176.796,24.806,153.994
C07948=1086.426,339.541,-90.916,176.799,24.811,153.994
C07949=1086.432,339.788,-90.950,176.802,24.815,153.995
C07950=1086.438,340.037,-90.984,176.805,24.820,153.996
C07951=1086.444,340.284,-91.018,176.808,24.824,153.996
C07952=1086.449,340.532,-91.052,176.812,24.829,153.997
C07953=1086.455,340.779,-91.086,176.814,24.834,153.998
C07954=1086.461,341.027,-91.120,176.817,24.838,153.998
C07955=1086.467,341.275,-91.154,176.821,24.844,153.999
C07956=1086.472,341.522,-91.188,176.824,24.848,154.000
C07957=1086.478,341.770,-91.222,176.826,24.852,154.001
C07958=1086.484,342.018,-91.256,176.830,24.857,154.001
C07959=1086.490,342.266,-91.290,176.833,24.862,154.002
C07960=1086.496,342.513,-91.324,176.836,24.866,154.003
C07961=1086.502,342.760,-91.358,176.839,24.871,154.003
C07962=1086.509,343.008,-91.393,176.842,24.875,154.004
C07963=1086.518,343.403,-91.447,176.847,24.883,154.005
C07964=1086.527,343.799,-91.502,176.852,24.890,154.006
C07965=1086.537,344.194,-91.557,176.857,24.898,154.007
C07966=1086.546,344.589,-91.611,176.862,24.906,154.008
C07967=1086.552,344.836,-91.646,176.865,24.910,154.009
C07968=1086.558,345.084,-91.680,176.868,24.915,154.010
C07969=1086.564,345.332,-91.714,176.871,24.920,154.011
C07970=1086.570,345.579,-91.748,176.875,24.925,154.011
C07971=1086.576,345.827,-91.783,176.877,24.930,154.012
C07972=1086.581,346.075,-91.817,176.880,24.934,154.013
C07973=1086.587,346.322,-91.851,176.884,24.939,154.014
C07974=1086.593,346.570,-91.886,176.886,24.944,154.014
C07975=1086.599,346.817,-91.920,176.890,24.949,154.015
C07976=1086.605,347.064,-91.955,176.893,24.953,154.016
C07977=1086.611,347.312,-91.990,176.896,24.959,154.017
C07978=1086.617,347.560,-92.024,176.899,24.963,154.017
C07979=1086.622,347.808,-92.059,176.902,24.968,154.018
C07980=1086.628,348.055,-92.094,176.906,24.973,154.019
C07981=1086.634,348.302,-92.128,176.908,24.978,154.020
C07982=1086.640,348.550,-92.163,176.912,24.983,154.020
C07983=1086.646,348.798,-92.197,176.915,24.988,154.021
C07984=1086.652,349.045,-92.233,176.918,24.993,154.022
C07985=1086.658,349.293,-92.267,176.921,24.997,154.022
C07986=1086.664,349.540,-92.301,176.924,25.002,154.023
C07987=1086.670,349.787,-92.337,176.927,25.007,154.024
C07988=1086.676,350.035,-92.371,176.930,25.012,154.025
C07989=1086.681,350.283,-92.406,176.933,25.017,154.026
C07990=1086.687,350.530,-92.441,176.936,25.022,154.026
C07991=1086.693,350.778,-92.476,176.940,25.027,154.027
C07992=1086.699,351.025,-92.510,176.943,25.032,154.028
C07993=1086.705,351.273,-92.545,176.946,25.037,154.029
C07994=1086.711,351.520,-92.580,176.949,25.042,154.029
C07995=1086.717,351.768,-92.615,176.952,25.047,154.030
C07996=1086.723,352.015,-92.650,176.955,25.052,154.031
C07997=1086.729,352.263,-92.685,176.959,25.057,154.032
C07998=1086.735,352.510,-92.720,176.961,25.062,154.033
C07999=1086.741,352.758,-92.755,176.965,25.067,154.033
C08000=1086.747,353.005,-92.790,176.968,25.072,154.034
C08001=1086.753,353.252,-92.825,176.971,25.077,154.035
C08002=1086.759,353.500,-92.860,176.974,25.082,154.036
C08003=1086.765,353.747,-92.895,176.978,25.088,154.037
C08004=1086.771,353.995,-92.931,176.980,25.092,154.037
C08005=1086.776,354.242,-92.965,176.984,25.098,154.038
C08006=1086.783,354.490,-93.001,176.986,25.103,154.039
C08007=1086.788,354.737,-93.036,176.990,25.108,154.040
C08008=1086.794,354.985,-93.071,176.993,25.113,154.041
C08009=1086.800,355.232,-93.106,176.996,25.118,154.041
C08010=1086.806,355.479,-93.141,176.999,25.123,154.042
C08011=1086.812,355.727,-93.177,177.002,25.129,154.043
C08012=1086.818,355.974,-93.213,177.005,25.134,154.044
C08013=1086.824,356.222,-93.247,177.009,25.139,154.045
C08014=1086.829,356.469,-93.282,177.011,25.144,154.046
C08015=1086.839,356.867,-93.340,177.017,25.153,154.047
C08016=1086.849,357.265,-93.396,177.022,25.161,154.048
C08017=1086.859,357.663,-93.453,177.026,25.169,154.050
C08018=1086.868,358.061,-93.510,177.031,25.177,154.051
C08019=1086.874,358.309,-93.546,177.035,25.183,154.052
C08020=1086.879,358.556,-93.582,177.038,25.188,154.053
C08021=1086.886,358.803,-93.617,177.041,25.193,154.054
C08022=1086.892,359.051,-93.652,177.045,25.199,154.054
C08023=1086.898,359.299,-93.688,177.047,25.204,154.055
C08024=1086.904,359.546,-93.724,177.051,25.210,154.056
C08025=1086.910,359.793,-93.759,177.053,25.214,154.057
C08026=1086.916,360.041,-93.795,177.057,25.220,154.058
C08027=1086.922,360.287,-93.830,177.061,25.225,154.059
C08028=1086.928,360.535,-93.866,177.063,25.231,154.060
C08029=1086.934,360.782,-93.902,177.067,25.237,154.061
C08030=1086.940,361.030,-93.938,177.069,25.241,154.061
C08031=1086.946,361.277,-93.973,177.073,25.247,154.062
C08032=1086.952,361.525,-94.009,177.076,25.253,154.063
C08033=1086.958,361.772,-94.045,177.079,25.258,154.064
C08034=1086.964,362.019,-94.081,177.082,25.264,154.065
C08035=1086.970,362.266,-94.116,177.085,25.269,154.066
C08036=1086.976,362.513,-94.153,177.089,25.274,154.067
C08037=1086.982,362.761,-94.188,177.092,25.280,154.068
C08038=1086.988,363.009,-94.224,177.095,25.285,154.069
C08039=1086.994,363.255,-94.260,177.098,25.291,154.070
C08040=1087.000,363.503,-94.296,177.101,25.296,154.070
C08041=1087.006,363.750,-94.332,177.104,25.302,154.071
C08042=1087.012,363.997,-94.368,177.108,25.308,154.072
C08043=1087.018,364.245,-94.404,177.110,25.313,154.073
C08044=1087.024,364.491,-94.440,177.114,25.318,154.074
C08045=1087.030,364.739,-94.476,177.117,25.324,154.075
C08046=1087.035,364.987,-94.513,177.120,25.329,154.076
C08047=1087.041,365.234,-94.549,177.123,25.335,154.077
C08048=1087.048,365.481,-94.585,177.127,25.341,154.078
C08049=1087.054,365.729,-94.621,177.130,25.346,154.079
C08050=1087.060,365.976,-94.657,177.133,25.352,154.080
C08051=1087.066,366.223,-94.692,177.136,25.358,154.081
C08052=1087.071,366.470,-94.730,177.139,25.363,154.082
C08053=1087.078,366.717,-94.766,177.142,25.369,154.083
C08054=1087.084,366.965,-94.802,177.146,25.375,154.084
C08055=1087.090,367.212,-94.838,177.148,25.381,154.085
C08056=1087.096,367.459,-94.875,177.152,25.386,154.086
C08057=1087.101,367.706,-94.911,177.155,25.392,154.087
C08058=1087.107,367.954,-94.947,177.158,25.398,154.088
C08059=1087.113,368.201,-94.984,177.161,25.404,154.088
C08060=1087.119,368.449,-95.020,177.165,25.410,154.090
C08061=1087.125,368.696,-95.056,177.167,25.415,154.090
C08062=1087.131,368.943,-95.093,177.171,25.421,154.092
C08063=1087.137,369.190,-95.130,177.174,25.427,154.092
C08064=1087.144,369.437,-95.166,177.177,25.433,154.094
C08065=1087.149,369.684,-95.203,177.180,25.438,154.094
C08066=1087.155,369.932,-95.239,177.184,25.445,154.096
C08067=1087.166,370.345,-95.300,177.189,25.454,154.097
C08068=1087.176,370.759,-95.362,177.195,25.464,154.099
C08069=1087.185,371.173,-95.423,177.200,25.474,154.101
C08070=1087.196,371.586,-95.484,177.204,25.483,154.102
C08071=1087.202,371.834,-95.521,177.208,25.490,154.103
C08072=1087.208,372.081,-95.558,177.211,25.496,154.104
C08073=1087.214,372.328,-95.594,177.215,25.502,154.105
C08074=1087.220,372.575,-95.631,177.217,25.507,154.106
C08075=1087.226,372.822,-95.668,177.221,25.513,154.107
C08076=1087.232,373.070,-95.705,177.224,25.520,154.108
C08077=1087.238,373.317,-95.741,177.227,25.526,154.110
C08078=1087.245,373.563,-95.778,177.230,25.532,154.111
C08079=1087.251,373.811,-95.815,177.233,25.538,154.112
C08080=1087.257,374.058,-95.852,177.237,25.544,154.113
C08081=1087.262,374.305,-95.889,177.240,25.550,154.114
C08082=1087.268,374.552,-95.926,177.243,25.556,154.115
C08083=1087.275,374.799,-95.963,177.246,25.562,154.116
C08084=1087.280,375.046,-96.000,177.249,25.568,154.117
C08085=1087.286,375.294,-96.037,177.253,25.575,154.118
C08086=1087.293,375.541,-96.075,177.256,25.581,154.119
C08087=1087.299,375.788,-96.112,177.259,25.587,154.120
C08088=1087.304,376.035,-96.149,177.262,25.593,154.121
C08089=1087.311,376.282,-96.186,177.265,25.599,154.123
C08090=1087.317,376.529,-96.223,177.269,25.606,154.124
C08091=1087.322,376.777,-96.260,177.272,25.612,154.125
C08092=1087.329,377.023,-96.297,177.275,25.618,154.126
C08093=1087.334,377.270,-96.334,177.278,25.624,154.127
C08094=1087.340,377.517,-96.372,177.281,25.631,154.128
C08095=1087.347,377.765,-96.409,177.285,25.637,154.129
C08096=1087.353,378.012,-96.446,177.288,25.643,154.130
C08097=1087.359,378.259,-96.483,177.291,25.650,154.131
C08098=1087.365,378.506,-96.521,177.295,25.656,154.133
C08099=1087.371,378.752,-96.558,177.297,25.662,154.134
C08100=1087.377,379.000,-96.595,177.300,25.669,154.135
C08101=1087.383,379.247,-96.634,177.304,25.675,154.136
C08102=1087.390,379.494,-96.670,177.307,25.681,154.137
C08103=1087.396,379.741,-96.708,177.310,25.688,154.138
C08104=1087.402,379.987,-96.746,177.314,25.695,154.140
C08105=1087.407,380.235,-96.783,177.317,25.701,154.141
C08106=1087.414,380.482,-96.821,177.320,25.707,154.142
C08107=1087.420,380.729,-96.858,177.323,25.714,154.143
C08108=1087.426,380.975,-96.896,177.326,25.720,154.144
C08109=1087.432,381.224,-96.933,177.330,25.727,154.145
C08110=1087.438,381.470,-96.971,177.333,25.733,154.147
C08111=1087.445,381.717,-97.008,177.336,25.739,154.148
C08112=1087.451,381.963,-97.046,177.340,25.746,154.149
C08113=1087.457,382.211,-97.084,177.343,25.753,154.150
C08114=1087.463,382.458,-97.121,177.346,25.759,154.151
C08115=1087.469,382.705,-97.159,177.349,25.766,154.152
C08116=1087.475,382.952,-97.197,177.352,25.773,154.154
C08117=1087.481,383.199,-97.234,177.355,25.779,154.155
C08118=1087.487,383.446,-97.272,177.359,25.786,154.156
C08119=1087.496,383.796,-97.326,177.363,25.795,154.158
C08120=1087.504,384.147,-97.381,177.368,25.805,154.160
C08121=1087.513,384.497,-97.434,177.372,25.815,154.161
C08122=1087.522,384.847,-97.487,177.377,25.824,154.163
C08123=1087.528,385.094,-97.526,177.380,25.831,154.164
C08124=1087.534,385.341,-97.564,177.383,25.838,154.166
C08125=1087.540,385.588,-97.602,177.387,25.845,154.167
C08126=1087.546,385.836,-97.640,177.390,25.852,154.168
C08127=1087.552,386.082,-97.678,177.393,25.858,154.169
C08128=1087.558,386.329,-97.716,177.396,25.865,154.171
C08129=1087.565,386.576,-97.755,177.400,25.872,154.172
C08130=1087.571,386.823,-97.792,177.403,25.879,154.173
C08131=1087.577,387.070,-97.831,177.406,25.886,154.175
C08132=1087.583,387.317,-97.868,177.409,25.893,154.176
C08133=1087.589,387.563,-97.907,177.413,25.900,154.177
C08134=1087.595,387.811,-97.946,177.416,25.907,154.178
C08135=1087.601,388.057,-97.983,177.419,25.914,154.180
C08136=1087.608,388.304,-98.022,177.422,25.921,154.181
C08137=1087.614,388.551,-98.060,177.426,25.928,154.182
C08138=1087.620,388.798,-98.099,177.429,25.935,154.184
C08139=1087.626,389.045,-98.136,177.432,25.942,154.185
C08140=1087.632,389.292,-98.175,177.435,25.949,154.186
C08141=1087.638,389.538,-98.214,177.439,25.956,154.188
C08142=1087.645,389.786,-98.252,177.442,25.963,154.189
C08143=1087.651,390.032,-98.290,177.445,25.970,154.190
C08144=1087.657,390.279,-98.328,177.448,25.977,154.192
C08145=1087.663,390.526,-98.367,177.451,25.985,154.193
C08146=1087.670,390.773,-98.406,177.455,25.992,154.194
C08147=1087.676,391.020,-98.444,177.458,25.999,154.196
C08148=1087.682,391.266,-98.483,177.462,26.006,154.197
C08149=1087.689,391.514,-98.521,177.465,26.013,154.198
C08150=1087.694,391.760,-98.560,177.469,26.021,154.200
C08151=1087.701,392.007,-98.599,177.472,26.028,154.201
C08152=1087.708,392.254,-98.637,177.475,26.035,154.202
C08153=1087.713,392.501,-98.676,177.478,26.043,154.204
C08154=1087.720,392.748,-98.715,177.481,26.050,154.205
C08155=1087.725,392.994,-98.754,177.484,26.057,154.207
C08156=1087.732,393.242,-98.792,177.488,26.065,154.208
C08157=1087.738,393.489,-98.832,177.491,26.072,154.210
C08158=1087.744,393.735,-98.870,177.494,26.079,154.211
C08159=1087.750,393.982,-98.909,177.497,26.086,154.212
C08160=1087.757,394.229,-98.948,177.501,26.094,154.214
C08161=1087.763,394.475,-98.987,177.504,26.102,154.215
C08162=1087.769,394.722,-99.026,177.508,26.109,154.217
C08163=1087.778,395.060,-99.079,177.512,26.119,154.219
C08164=1087.786,395.399,-99.133,177.517,26.130,154.221
C08165=1087.795,395.736,-99.187,177.521,26.140,154.223
C08166=1087.803,396.074,-99.240,177.525,26.151,154.225
C08167=1087.809,396.321,-99.279,177.529,26.158,154.226
C08168=1087.816,396.568,-99.318,177.532,26.166,154.228
C08169=1087.822,396.814,-99.357,177.535,26.173,154.229
C08170=1087.828,397.062,-99.397,177.539,26.182,154.231
C08171=1087.834,397.289,-99.433,177.541,26.188,154.232
C08172=1087.840,397.517,-99.469,177.544,26.196,154.233
C08173=1087.845,397.744,-99.505,177.548,26.203,154.235
C08174=1087.851,397.972,-99.541,177.551,26.210,154.236
C08175=1087.857,398.200,-99.578,177.553,26.217,154.238
C08176=1087.863,398.428,-99.614,177.556,26.224,154.239
C08177=1087.868,398.655,-99.650,177.560,26.232,154.240
C08178=1087.874,398.882,-99.686,177.563,26.239,154.242
C08179=1087.880,399.129,-99.726,177.566,26.247,154.243
C08180=1087.886,399.377,-99.765,177.569,26.255,154.245
C08181=1087.893,399.623,-99.805,177.572,26.263,154.246
C08182=1087.899,399.870,-99.844,177.576,26.271,154.248
C08183=1087.905,400.116,-99.884,177.579,26.279,154.250
C08184=1087.911,400.363,-99.924,177.582,26.287,154.251
C08185=1087.917,400.610,-99.963,177.586,26.295,154.253
C08186=1087.924,400.857,-100.003,177.590,26.303,154.254
C08187=1087.930,401.104,-100.043,177.593,26.311,154.256
C08188=1087.937,401.350,-100.082,177.596,26.319,154.257
C08189=1087.943,401.597,-100.122,177.599,26.327,154.259
C08190=1087.949,401.844,-100.162,177.603,26.335,154.261
C08191=1087.956,402.091,-100.201,177.606,26.343,154.262
C08192=1087.962,402.337,-100.241,177.609,26.352,154.264
C08193=1087.968,402.584,-100.281,177.613,26.360,154.266
C08194=1087.974,402.831,-100.321,177.616,26.368,154.267
C08195=1087.981,403.077,-100.361,177.619,26.376,154.269
C08196=1087.987,403.325,-100.400,177.623,26.384,154.270
C08197=1087.993,403.571,-100.441,177.626,26.393,154.272
C08198=1088.000,403.818,-100.481,177.629,26.401,154.274
C08199=1088.006,404.065,-100.520,177.633,26.409,154.275
C08200=1088.012,404.311,-100.560,177.636,26.418,154.277
C08201=1088.018,404.558,-100.600,177.639,26.426,154.279
C08202=1088.025,404.804,-100.641,177.643,26.435,154.280
C08203=1088.031,405.051,-100.680,177.646,26.443,154.282
C08204=1088.037,405.298,-100.720,177.649,26.451,154.284
C08205=1088.044,405.544,-100.760,177.653,26.460,154.286
C08206=1088.050,405.791,-100.800,177.656,26.469,154.287
C08207=1088.056,406.037,-100.841,177.659,26.477,154.289
C08208=1088.063,406.284,-100.881,177.663,26.486,154.291
C08209=1088.068,406.531,-100.921,177.666,26.494,154.293
C08210=1088.075,406.778,-100.962,177.670,26.503,154.294
C08211=1088.082,407.024,-101.002,177.673,26.511,154.296
C08212=1088.088,407.271,-101.042,177.677,26.521,154.298
C08213=1088.095,407.518,-101.082,177.680,26.529,154.299
C08214=1088.101,407.764,-101.123,177.683,26.538,154.301
C08215=1088.107,408.011,-101.163,177.687,26.546,154.303
C08216=1088.113,408.257,-101.203,177.690,26.555,154.305
C08217=1088.120,408.505,-101.244,177.694,26.564,154.307
C08218=1088.126,408.751,-101.285,177.697,26.573,154.308
C08219=1088.132,408.998,-101.325,177.701,26.582,154.310
C08220=1088.139,409.244,-101.366,177.703,26.591,154.312
C08221=1088.144,409.491,-101.406,177.707,26.600,154.314
C08222=1088.151,409.737,-101.447,177.710,26.609,154.316
C08223=1088.157,409.985,-101.488,177.714,26.618,154.317
C08224=1088.164,410.231,-101.529,177.717,26.627,154.319
C08225=1088.170,410.477,-101.569,177.721,26.636,154.321
C08226=1088.176,410.724,-101.609,177.724,26.645,154.323
C08227=1088.182,410.952,-101.648,177.727,26.653,154.325
C08228=1088.188,411.180,-101.686,177.731,26.662,154.326
C08229=1088.194,411.409,-101.723,177.734,26.670,154.328
C08230=1088.200,411.637,-101.761,177.737,26.679,154.330
C08231=1088.206,411.864,-101.798,177.740,26.687,154.332
C08232=1088.211,412.093,-101.836,177.743,26.696,154.333
C08233=1088.217,412.321,-101.874,177.746,26.704,154.335
C08234=1088.224,412.549,-101.912,177.750,26.713,154.337
C08235=1088.230,412.796,-101.952,177.753,26.722,154.339
C08236=1088.236,413.043,-101.994,177.757,26.731,154.341
C08237=1088.243,413.289,-102.034,177.760,26.741,154.343
C08238=1088.249,413.536,-102.076,177.764,26.750,154.345
C08239=1088.256,413.782,-102.117,177.768,26.759,154.346
C08240=1088.262,414.029,-102.158,177.771,26.769,154.348
C08241=1088.269,414.275,-102.199,177.774,26.778,154.350
C08242=1088.275,414.522,-102.241,177.778,26.788,154.352
C08243=1088.282,414.769,-102.281,177.781,26.797,154.354
C08244=1088.288,415.015,-102.323,177.785,26.807,154.356
C08245=1088.295,415.261,-102.363,177.789,26.816,154.358
C08246=1088.301,415.508,-102.405,177.792,26.826,154.360
C08247=1088.308,415.754,-102.446,177.796,26.835,154.362
C08248=1088.314,416.001,-102.488,177.799,26.845,154.364
C08249=1088.320,416.248,-102.529,177.802,26.855,154.366
C08250=1088.327,416.494,-102.570,177.806,26.865,154.368
C08251=1088.333,416.740,-102.611,177.810,26.874,154.370
C08252=1088.340,416.987,-102.653,177.814,26.884,154.372
C08253=1088.346,417.233,-102.695,177.816,26.894,154.374
C08254=1088.353,417.480,-102.736,177.820,26.904,154.376
C08255=1088.359,417.726,-102.778,177.824,26.914,154.378
C08256=1088.366,417.972,-102.820,177.828,26.924,154.380
C08257=1088.372,418.219,-102.861,177.831,26.933,154.383
C08258=1088.379,418.465,-102.903,177.834,26.943,154.385
C08259=1088.385,418.711,-102.944,177.838,26.953,154.387
C08260=1088.392,418.958,-102.986,177.842,26.963,154.389
C08261=1088.398,419.205,-103.027,177.846,26.974,154.391
C08262=1088.404,419.451,-103.070,177.849,26.984,154.393
C08263=1088.411,419.698,-103.112,177.852,26.994,154.395
C08264=1088.418,419.944,-103.152,177.856,27.004,154.397
C08265=1088.424,420.190,-103.195,177.860,27.015,154.400
C08266=1088.430,420.436,-103.236,177.864,27.024,154.402
C08267=1088.437,420.683,-103.278,177.867,27.035,154.404
C08268=1088.444,420.929,-103.321,177.871,27.045,154.406
C08269=1088.450,421.176,-103.362,177.874,27.055,154.408
C08270=1088.457,421.422,-103.405,177.878,27.065,154.410
C08271=1088.464,421.668,-103.446,177.881,27.076,154.412
C08272=1088.470,421.914,-103.488,177.885,27.086,154.415
C08273=1088.477,422.161,-103.530,177.889,27.097,154.417
C08274=1088.484,422.407,-103.573,177.893,27.107,154.419
C08275=1088.490,422.653,-103.614,177.896,27.118,154.421
C08276=1088.496,422.900,-103.657,177.900,27.129,154.424
C08277=1088.503,423.146,-103.699,177.904,27.139,154.426
C08278=1088.509,423.393,-103.742,177.907,27.150,154.428
C08279=1088.515,423.639,-103.784,177.911,27.161,154.430
C08280=1088.522,423.885,-103.826,177.915,27.171,154.433
C08281=1088.529,424.132,-103.868,177.919,27.182,154.435
C08282=1088.535,424.378,-103.910,177.922,27.193,154.437
C08283=1088.542,424.614,-103.951,177.925,27.203,154.439
C08284=1088.547,424.849,-103.992,177.929,27.213,154.442
C08285=1088.554,425.085,-104.032,177.933,27.224,154.444
C08286=1088.561,425.322,-104.073,177.936,27.235,154.446
C08287=1088.567,425.557,-104.114,177.939,27.245,154.448
C08288=1088.573,425.793,-104.154,177.943,27.255,154.451
C08289=1088.579,426.029,-104.195,177.947,27.266,154.453
C08290=1088.586,426.264,-104.236,177.951,27.276,154.455
C08291=1088.593,426.511,-104.279,177.954,27.288,154.458
C08292=1088.599,426.757,-104.322,177.958,27.299,154.460
C08293=1088.606,427.004,-104.365,177.961,27.310,154.462
C08294=1088.613,427.250,-104.407,177.965,27.321,154.465
C08295=1088.619,427.495,-104.449,177.969,27.332,154.467
C08296=1088.625,427.742,-104.492,177.972,27.343,154.470
C08297=1088.632,427.988,-104.535,177.976,27.355,154.472
C08298=1088.639,428.234,-104.578,177.980,27.366,154.474
C08299=1088.646,428.480,-104.621,177.984,27.378,154.477
C08300=1088.652,428.727,-104.664,177.988,27.389,154.479
C08301=1088.659,428.973,-104.706,177.992,27.400,154.482
C08302=1088.666,429.219,-104.750,177.995,27.412,154.484
C08303=1088.672,429.465,-104.793,177.999,27.423,154.487
C08304=1088.679,429.711,-104.836,178.003,27.435,154.489
C08305=1088.685,429.958,-104.879,178.007,27.447,154.492
C08306=1088.692,430.204,-104.922,178.011,27.458,154.494
C08307=1088.699,430.450,-104.966,178.014,27.470,154.497
C08308=1088.706,430.696,-105.009,178.018,27.481,154.499
C08309=1088.713,430.942,-105.051,178.022,27.493,154.502
C08310=1088.719,431.188,-105.095,178.026,27.505,154.505
C08311=1088.726,431.434,-105.138,178.030,27.517,154.507
C08312=1088.732,431.680,-105.182,178.033,27.529,154.510
C08313=1088.740,431.926,-105.225,178.037,27.541,154.512
C08314=1088.746,432.172,-105.268,178.041,27.553,154.515
C08315=1088.753,432.418,-105.311,178.045,27.565,154.518
C08316=1088.759,432.664,-105.355,178.049,27.577,154.520
C08317=1088.765,432.911,-105.398,178.052,27.589,154.523
C08318=1088.773,433.156,-105.441,178.057,27.601,154.526
C08319=1088.779,433.402,-105.485,178.060,27.613,154.528
C08320=1088.785,433.648,-105.529,178.064,27.626,154.531
C08321=1088.793,433.894,-105.573,178.069,27.638,154.534
C08322=1088.800,434.140,-105.617,178.072,27.650,154.536
C08323=1088.806,434.386,-105.660,178.076,27.662,154.539
C08324=1088.813,434.632,-105.704,178.080,27.675,154.542
C08325=1088.820,434.878,-105.748,178.084,27.687,154.545
C08326=1088.826,435.124,-105.791,178.087,27.700,154.547
C08327=1088.832,435.370,-105.835,178.092,27.713,154.550
C08328=1088.840,435.616,-105.879,178.095,27.725,154.553
C08329=1088.847,435.862,-105.923,178.099,27.737,154.556
C08330=1088.853,436.108,-105.967,178.103,27.750,154.558
C08331=1088.860,436.354,-106.011,178.107,27.763,154.561
C08332=1088.866,436.600,-106.055,178.111,27.776,154.564
C08333=1088.874,436.846,-106.099,178.115,27.788,154.567
C08334=1088.881,437.091,-106.143,178.119,27.801,154.570
C08335=1088.887,437.337,-106.187,178.123,27.814,154.573
C08336=1088.894,437.584,-106.231,178.127,27.827,154.576
C08337=1088.901,437.829,-106.276,178.131,27.840,154.578
C08338=1088.907,438.075,-106.320,178.135,27.853,154.581
C08339=1088.916,438.371,-106.372,178.140,27.868,154.585
C08340=1088.925,438.667,-106.426,178.145,27.884,154.588
C08341=1088.933,438.962,-106.479,178.150,27.900,154.592
C08342=1088.941,439.258,-106.533,178.155,27.916,154.595
C08343=1088.948,439.504,-106.577,178.158,27.930,154.598
C08344=1088.955,439.750,-106.622,178.163,27.943,154.601
C08345=1088.962,439.995,-106.666,178.166,27.956,154.604
C08346=1088.969,440.242,-106.710,178.171,27.970,154.607
C08347=1088.976,440.487,-106.755,178.174,27.983,154.610
C08348=1088.983,440.733,-106.800,178.179,27.996,154.613
C08349=1088.990,440.978,-106.844,178.183,28.010,154.617
C08350=1088.996,441.224,-106.888,178.186,28.024,154.620
C08351=1089.003,441.471,-106.933,178.191,28.038,154.623
C08352=1089.010,441.716,-106.978,178.194,28.051,154.626
C08353=1089.017,441.962,-107.023,178.199,28.065,154.629
C08354=1089.023,442.208,-107.068,178.203,28.079,154.632
C08355=1089.031,442.454,-107.113,178.207,28.092,154.635
C08356=1089.037,442.699,-107.157,178.211,28.107,154.638
C08357=1089.045,442.945,-107.202,178.216,28.120,154.641
C08358=1089.052,443.190,-107.247,178.219,28.134,154.645
C08359=1089.058,443.436,-107.293,178.224,28.149,154.648
C08360=1089.065,443.681,-107.338,178.228,28.163,154.651
C08361=1089.072,443.928,-107.383,178.232,28.177,154.654
C08362=1089.080,444.174,-107.428,178.236,28.191,154.657
C08363=1089.086,444.419,-107.473,178.240,28.206,154.661
C08364=1089.093,444.665,-107.518,178.245,28.220,154.664
C08365=1089.100,444.910,-107.563,178.248,28.234,154.667
C08366=1089.107,445.156,-107.608,178.252,28.248,154.671
C08367=1089.114,445.402,-107.654,178.255,28.263,154.674
C08368=1089.122,445.648,-107.699,178.259,28.277,154.677
C08369=1089.128,445.893,-107.745,178.262,28.292,154.681
C08370=1089.135,446.139,-107.790,178.265,28.306,154.684
C08371=1089.143,446.384,-107.835,178.268,28.320,154.687
C08372=1089.149,446.630,-107.881,178.271,28.334,154.691
C08373=1089.157,446.876,-107.926,178.272,28.348,154.694
C08374=1089.163,447.122,-107.972,178.275,28.363,154.698
C08375=1089.171,447.367,-108.017,178.277,28.377,154.701
C08376=1089.177,447.612,-108.063,178.279,28.391,154.704
C08377=1089.184,447.858,-108.108,178.280,28.405,154.708
C08378=1089.191,448.104,-108.154,178.282,28.419,154.711
C08379=1089.199,448.350,-108.200,178.283,28.434,154.715
C08380=1089.206,448.596,-108.246,178.284,28.448,154.718
C08381=1089.213,448.841,-108.291,178.286,28.462,154.722
C08382=1089.220,449.086,-108.337,178.286,28.476,154.725
C08383=1089.227,449.332,-108.383,178.287,28.490,154.729
C08384=1089.234,449.577,-108.428,178.287,28.504,154.732
C08385=1089.242,449.822,-108.474,178.288,28.518,154.736
C08386=1089.252,450.069,-108.518,178.289,28.531,154.739
C08387=1088.872,450.060,-108.710,178.247,28.724,154.792
C08388=1088.862,449.813,-108.665,178.246,28.711,154.789
C08389=1088.853,449.568,-108.620,178.246,28.698,154.785
C08390=1088.847,449.323,-108.574,178.245,28.684,154.782
C08391=1088.839,449.078,-108.528,178.244,28.670,154.778
C08392=1088.832,448.832,-108.482,178.244,28.655,154.775
C08393=1088.825,448.586,-108.437,178.242,28.641,154.771
C08394=1088.818,448.340,-108.391,178.241,28.627,154.768
C08395=1088.811,448.096,-108.345,178.239,28.613,154.764
C08396=1088.804,447.850,-108.299,178.238,28.599,154.761
C08397=1088.797,447.604,-108.254,178.236,28.584,154.757
C08398=1088.790,447.358,-108.208,178.234,28.570,154.754
C08399=1088.782,447.113,-108.162,178.232,28.556,154.750
C08400=1088.775,446.867,-108.117,178.229,28.541,154.747
C08401=1088.769,446.621,-108.072,178.228,28.527,154.744
C08402=1088.761,446.376,-108.026,178.225,28.513,154.740
C08403=1088.754,446.130,-107.980,178.221,28.499,154.737
C08404=1088.747,445.884,-107.935,178.219,28.484,154.733
C08405=1088.740,445.639,-107.889,178.215,28.470,154.730
C08406=1088.733,445.393,-107.844,178.212,28.455,154.727
C08407=1088.726,445.148,-107.798,178.208,28.441,154.723
C08408=1088.720,444.902,-107.753,178.204,28.427,154.720
C08409=1088.712,444.656,-107.708,178.200,28.413,154.717
C08410=1088.705,444.411,-107.663,178.196,28.398,154.713
C08411=1088.699,444.165,-107.617,178.192,28.384,154.710
C08412=1088.691,443.919,-107.572,178.187,28.369,154.707
C08413=1088.684,443.673,-107.527,178.184,28.356,154.704
C08414=1088.677,443.428,-107.482,178.179,28.341,154.701
C08415=1088.670,443.182,-107.437,178.175,28.327,154.697
C08416=1088.664,442.936,-107.392,178.170,28.313,154.694
C08417=1088.656,442.691,-107.347,178.167,28.299,154.691
C08418=1088.649,442.445,-107.302,178.162,28.285,154.688
C08419=1088.642,442.199,-107.257,178.158,28.271,154.685
C08420=1088.635,441.953,-107.211,178.154,28.257,154.681
C08421=1088.629,441.708,-107.167,178.149,28.243,154.678
C08422=1088.621,441.462,-107.122,178.146,28.229,154.675
C08423=1088.614,441.216,-107.077,178.141,28.216,154.672
C08424=1088.607,440.970,-107.032,178.137,28.202,154.669
C08425=1088.600,440.725,-106.988,178.133,28.188,154.666
C08426=1088.593,440.478,-106.944,178.128,28.175,154.663
C08427=1088.587,440.233,-106.899,178.125,28.162,154.660
C08428=1088.580,439.988,-106.855,178.120,28.148,154.657
C08429=1088.573,439.742,-106.810,178.117,28.135,154.654
C08430=1088.566,439.496,-106.766,178.112,28.121,154.651
C08431=1088.559,439.249,-106.721,178.109,28.108,154.648
C08432=1088.551,438.967,-106.670,178.103,28.093,154.645
C08433=1088.543,438.685,-106.619,178.099,28.078,154.641
C08434=1088.535,438.402,-106.568,178.094,28.062,154.638
C08435=1088.527,438.120,-106.517,178.090,28.048,154.634
C08436=1088.520,437.874,-106.473,178.085,28.034,154.632
C08437=1088.513,437.628,-106.428,178.081,28.022,154.629
C08438=1088.506,437.382,-106.384,178.077,28.008,154.626
C08439=1088.500,437.137,-106.340,178.073,27.996,154.623
C08440=1088.493,436.890,-106.296,178.070,27.983,154.620
C08441=1088.485,436.644,-106.252,178.065,27.970,154.617
C08442=1088.479,436.399,-106.208,178.061,27.957,154.614
C08443=1088.472,436.153,-106.164,178.057,27.944,154.612
C08444=1088.465,435.906,-106.120,178.053,27.932,154.609
C08445=1088.459,435.661,-106.075,178.050,27.919,154.606
C08446=1088.451,435.415,-106.032,178.045,27.907,154.603
C08447=1088.445,435.169,-105.988,178.041,27.894,154.600
C08448=1088.438,434.923,-105.944,178.037,27.881,154.598
C08449=1088.431,434.677,-105.900,178.033,27.869,154.595
C08450=1088.424,434.431,-105.857,178.029,27.856,154.592
C08451=1088.418,434.185,-105.813,178.025,27.844,154.589
C08452=1088.411,433.939,-105.769,178.021,27.832,154.587
C08453=1088.405,433.693,-105.725,178.017,27.819,154.584
C08454=1088.398,433.447,-105.682,178.014,27.807,154.581
C08455=1088.391,433.201,-105.638,178.009,27.795,154.579
C08456=1088.384,432.955,-105.594,178.005,27.783,154.576
C08457=1088.377,432.709,-105.551,178.002,27.770,154.573
C08458=1088.371,432.463,-105.507,177.997,27.758,154.570
C08459=1088.364,432.217,-105.464,177.994,27.746,154.568
C08460=1088.358,431.971,-105.420,177.990,27.734,154.565
C08461=1088.350,431.725,-105.377,177.986,27.722,154.563
C08462=1088.344,431.479,-105.333,177.982,27.710,154.560
C08463=1088.337,431.233,-105.291,177.978,27.699,154.557
C08464=1088.331,430.987,-105.247,177.974,27.686,154.555
C08465=1088.323,430.741,-105.203,177.971,27.675,154.552
C08466=1088.317,430.494,-105.160,177.967,27.663,154.550
C08467=1088.310,430.248,-105.117,177.962,27.651,154.547
C08468=1088.304,430.002,-105.074,177.958,27.640,154.545
C08469=1088.296,429.756,-105.031,177.955,27.628,154.542
C08470=1088.291,429.510,-104.988,177.951,27.616,154.539
C08471=1088.284,429.265,-104.944,177.947,27.605,154.537
C08472=1088.278,429.018,-104.901,177.944,27.593,154.534
C08473=1088.270,428.772,-104.858,177.940,27.582,154.532
C08474=1088.264,428.526,-104.816,177.935,27.570,154.530
C08475=1088.257,428.279,-104.772,177.932,27.558,154.527
C08476=1088.250,428.034,-104.729,177.928,27.547,154.525
C08477=1088.243,427.787,-104.687,177.924,27.536,154.522
C08478=1088.237,427.541,-104.644,177.920,27.525,154.520
C08479=1088.230,427.295,-104.601,177.917,27.514,154.517
C08480=1088.224,427.048,-104.558,177.913,27.502,154.515
C08481=1088.216,426.803,-104.515,177.909,27.491,154.512
C08482=1088.210,426.556,-104.473,177.905,27.480,154.510
C08483=1088.203,426.310,-104.430,177.902,27.469,154.508
C08484=1088.197,426.074,-104.389,177.898,27.458,154.505
C08485=1088.190,425.837,-104.348,177.894,27.448,154.503
C08486=1088.184,425.601,-104.308,177.890,27.437,154.501
C08487=1088.178,425.364,-104.266,177.886,27.426,154.499
C08488=1088.172,425.128,-104.226,177.883,27.416,154.496
C08489=1088.165,424.892,-104.185,177.880,27.406,154.494
C08490=1088.159,424.655,-104.144,177.876,27.395,154.492
C08491=1088.153,424.418,-104.103,177.872,27.384,154.490
C08492=1088.146,424.172,-104.061,177.868,27.373,154.487
C08493=1088.139,423.926,-104.018,177.865,27.363,154.485
C08494=1088.133,423.679,-103.976,177.862,27.352,154.483
C08495=1088.126,423.434,-103.934,177.858,27.342,154.480
C08496=1088.120,423.187,-103.892,177.854,27.331,154.478
C08497=1088.113,422.941,-103.849,177.850,27.320,154.476
C08498=1088.107,422.695,-103.807,177.847,27.309,154.474
C08499=1088.101,422.448,-103.765,177.843,27.299,154.471
C08500=1088.093,422.202,-103.723,177.839,27.289,154.469
C08501=1088.086,421.956,-103.680,177.835,27.278,154.467
C08502=1088.080,421.709,-103.639,177.831,27.267,154.465
C08503=1088.074,421.463,-103.596,177.828,27.257,154.463
C08504=1088.067,421.216,-103.554,177.824,27.246,154.460
C08505=1088.061,420.971,-103.512,177.821,27.236,154.458
C08506=1088.054,420.724,-103.470,177.817,27.226,154.456
C08507=1088.047,420.477,-103.428,177.813,27.216,154.454
C08508=1088.041,420.231,-103.386,177.809,27.205,154.452
C08509=1088.035,419.984,-103.344,177.806,27.195,154.449
C08510=1088.027,419.738,-103.302,177.802,27.185,154.447
C08511=1088.021,419.492,-103.261,177.799,27.175,154.445
C08512=1088.015,419.245,-103.219,177.795,27.165,154.443
C08513=1088.008,418.999,-103.177,177.791,27.155,154.441
C08514=1088.002,418.753,-103.135,177.787,27.145,154.439
C08515=1087.995,418.506,-103.094,177.783,27.135,154.437
C08516=1087.989,418.260,-103.053,177.781,27.124,154.435
C08517=1087.982,418.014,-103.010,177.777,27.114,154.433
C08518=1087.976,417.768,-102.969,177.773,27.104,154.430
C08519=1087.969,417.521,-102.927,177.769,27.094,154.428
C08520=1087.963,417.275,-102.886,177.766,27.085,154.426
C08521=1087.956,417.028,-102.844,177.762,27.075,154.424
C08522=1087.950,416.782,-102.803,177.759,27.065,154.422
C08523=1087.944,416.535,-102.761,177.755,27.055,154.420
C08524=1087.938,416.289,-102.719,177.752,27.046,154.418
C08525=1087.930,416.042,-102.678,177.748,27.036,154.416
C08526=1087.924,415.796,-102.637,177.744,27.026,154.414
C08527=1087.917,415.549,-102.595,177.741,27.016,154.412
C08528=1087.911,415.303,-102.554,177.737,27.007,154.410
C08529=1087.904,415.056,-102.513,177.733,26.997,154.408
C08530=1087.898,414.809,-102.472,177.730,26.988,154.406
C08531=1087.891,414.563,-102.431,177.726,26.978,154.404
C08532=1087.885,414.317,-102.389,177.723,26.968,154.402
C08533=1087.878,414.070,-102.348,177.720,26.959,154.400
C08534=1087.872,413.823,-102.307,177.716,26.950,154.398
C08535=1087.865,413.577,-102.266,177.712,26.940,154.396
C08536=1087.859,413.330,-102.225,177.709,26.931,154.394
C08537=1087.852,413.085,-102.184,177.705,26.921,154.393
C08538=1087.846,412.837,-102.143,177.702,26.912,154.391
C08539=1087.839,412.591,-102.102,177.698,26.903,154.389
C08540=1087.834,412.362,-102.064,177.695,26.894,154.387
C08541=1087.827,412.133,-102.025,177.692,26.885,154.385
C08542=1087.821,411.905,-101.988,177.688,26.877,154.383
C08543=1087.816,411.676,-101.950,177.685,26.869,154.382
C08544=1087.810,411.448,-101.912,177.682,26.860,154.380
C08545=1087.804,411.218,-101.874,177.678,26.852,154.378
C08546=1087.798,410.990,-101.836,177.675,26.843,154.376
C08547=1087.792,410.761,-101.799,177.672,26.834,154.375
C08548=1087.785,410.514,-101.757,177.668,26.825,154.373
C08549=1087.779,410.268,-101.717,177.665,26.817,154.371
C08550=1087.773,410.021,-101.676,177.661,26.807,154.369
C08551=1087.767,409.775,-101.635,177.658,26.798,154.367
C08552=1087.760,409.528,-101.595,177.654,26.789,154.365
C08553=1087.754,409.281,-101.554,177.651,26.780,154.364
C08554=1087.748,409.034,-101.514,177.647,26.771,154.362
C08555=1087.741,408.789,-101.473,177.644,26.762,154.360
C08556=1087.735,408.542,-101.432,177.640,26.753,154.358
C08557=1087.729,408.295,-101.392,177.637,26.744,154.356
C08558=1087.722,408.048,-101.352,177.633,26.736,154.355
C08559=1087.716,407.801,-101.311,177.630,26.727,154.353
C08560=1087.710,407.555,-101.270,177.627,26.718,154.351
C08561=1087.703,407.309,-101.230,177.623,26.709,154.349
C08562=1087.697,407.062,-101.190,177.620,26.701,154.347
C08563=1087.691,406.815,-101.149,177.616,26.692,154.346
C08564=1087.684,406.568,-101.108,177.613,26.683,154.344
C08565=1087.678,406.322,-101.068,177.610,26.675,154.342
C08566=1087.671,406.075,-101.028,177.606,26.666,154.340
C08567=1087.665,405.829,-100.988,177.603,26.657,154.339
C08568=1087.659,405.582,-100.948,177.599,26.649,154.337
C08569=1087.653,405.335,-100.908,177.596,26.640,154.335
C08570=1087.647,405.088,-100.868,177.593,26.632,154.334
C08571=1087.641,404.842,-100.827,177.589,26.623,154.332
C08572=1087.634,404.595,-100.787,177.586,26.615,154.330
C08573=1087.628,404.349,-100.747,177.583,26.607,154.329
C08574=1087.621,404.101,-100.707,177.579,26.598,154.327
C08575=1087.615,403.854,-100.667,177.576,26.590,154.325
C08576=1087.608,403.608,-100.627,177.573,26.581,154.324
C08577=1087.602,403.361,-100.587,177.569,26.573,154.322
C08578=1087.596,403.115,-100.547,177.566,26.565,154.320
C08579=1087.590,402.868,-100.507,177.563,26.556,154.319
C08580=1087.583,402.621,-100.467,177.558,26.548,154.317
C08581=1087.577,402.374,-100.428,177.555,26.540,154.315
C08582=1087.570,402.128,-100.388,177.552,26.532,154.314
C08583=1087.564,401.881,-100.348,177.549,26.523,154.312
C08584=1087.558,401.634,-100.309,177.545,26.515,154.311
C08585=1087.551,401.388,-100.268,177.542,26.507,154.309
C08586=1087.545,401.140,-100.229,177.539,26.499,154.307
C08587=1087.539,400.894,-100.189,177.536,26.491,154.306
C08588=1087.533,400.647,-100.150,177.532,26.483,154.304
C08589=1087.527,400.401,-100.110,177.529,26.474,154.302
C08590=1087.521,400.154,-100.070,177.526,26.467,154.301
C08591=1087.514,399.908,-100.031,177.522,26.459,154.299
C08592=1087.508,399.661,-99.991,177.518,26.450,154.298
C08593=1087.501,399.413,-99.952,177.515,26.442,154.296
C08594=1087.495,399.167,-99.912,177.512,26.435,154.295
C08595=1087.489,398.920,-99.872,177.509,26.427,154.293
C08596=1087.483,398.692,-99.836,177.506,26.420,154.292
C08597=1087.477,398.464,-99.800,177.502,26.412,154.290
C08598=1087.472,398.236,-99.763,177.499,26.405,154.289
C08599=1087.466,398.008,-99.727,177.497,26.398,154.287
C08600=1087.460,397.779,-99.691,177.493,26.391,154.286
C08601=1087.454,397.551,-99.654,177.490,26.383,154.285
C08602=1087.448,397.323,-99.618,177.487,26.376,154.283
C08603=1087.443,397.095,-99.582,177.484,26.369,154.282
C08604=1087.436,396.848,-99.543,177.480,26.361,154.280
C08605=1087.430,396.602,-99.503,177.477,26.354,154.279
C08606=1087.424,396.355,-99.464,177.474,26.346,154.277
C08607=1087.417,396.108,-99.425,177.471,26.338,154.276
C08608=1087.411,395.861,-99.385,177.468,26.331,154.274
C08609=1087.405,395.614,-99.347,177.465,26.323,154.273
C08610=1087.399,395.368,-99.307,177.461,26.315,154.271
C08611=1087.393,395.121,-99.268,177.457,26.308,154.270
C08612=1087.386,394.874,-99.229,177.454,26.300,154.268
C08613=1087.381,394.627,-99.190,177.451,26.293,154.267
C08614=1087.374,394.381,-99.151,177.448,26.285,154.266
C08615=1087.368,394.134,-99.112,177.444,26.277,154.264
C08616=1087.361,393.886,-99.074,177.441,26.270,154.263
C08617=1087.356,393.640,-99.035,177.438,26.263,154.261
C08618=1087.349,393.393,-98.996,177.435,26.255,154.260
C08619=1087.344,393.146,-98.957,177.431,26.248,154.258
C08620=1087.337,392.900,-98.918,177.428,26.240,154.257
C08621=1087.330,392.653,-98.879,177.425,26.233,154.255
C08622=1087.325,392.406,-98.841,177.421,26.225,154.254
C08623=1087.318,392.159,-98.802,177.418,26.218,154.253
C08624=1087.312,391.912,-98.762,177.414,26.211,154.251
C08625=1087.306,391.666,-98.724,177.411,26.204,154.250
C08626=1087.299,391.418,-98.686,177.408,26.196,154.249
C08627=1087.294,391.172,-98.647,177.405,26.189,154.247
C08628=1087.287,390.924,-98.609,177.401,26.182,154.246
C08629=1087.280,390.677,-98.570,177.398,26.175,154.244
C08630=1087.274,390.431,-98.531,177.395,26.168,154.243
C08631=1087.268,390.184,-98.493,177.392,26.160,154.242
C08632=1087.262,389.937,-98.454,177.388,26.153,154.240
C08633=1087.256,389.690,-98.416,177.385,26.146,154.239
C08634=1087.249,389.443,-98.377,177.382,26.139,154.238
C08635=1087.243,389.196,-98.339,177.379,26.132,154.236
C08636=1087.237,388.949,-98.300,177.375,26.125,154.235
C08637=1087.231,388.703,-98.262,177.372,26.117,154.234
C08638=1087.224,388.456,-98.223,177.369,26.110,154.232
C08639=1087.218,388.209,-98.186,177.366,26.103,154.231
C08640=1087.212,387.962,-98.147,177.362,26.096,154.230
C08641=1087.206,387.715,-98.109,177.359,26.089,154.228
C08642=1087.200,387.468,-98.071,177.356,26.082,154.227
C08643=1087.194,387.222,-98.032,177.352,26.075,154.226
C08644=1087.188,386.975,-97.994,177.349,26.069,154.225
C08645=1087.181,386.727,-97.956,177.346,26.062,154.223
C08646=1087.175,386.481,-97.918,177.342,26.055,154.222
C08647=1087.169,386.234,-97.879,177.339,26.048,154.221
C08648=1087.163,385.987,-97.842,177.336,26.041,154.219
C08649=1087.157,385.740,-97.804,177.333,26.034,154.218
C08650=1087.151,385.493,-97.765,177.329,26.027,154.217
C08651=1087.145,385.246,-97.727,177.326,26.020,154.216
C08652=1087.139,385.025,-97.693,177.323,26.014,154.214
C08653=1087.133,384.803,-97.659,177.320,26.008,154.213
C08654=1087.128,384.582,-97.625,177.317,26.002,154.212
C08655=1087.123,384.361,-97.591,177.314,25.995,154.211
C08656=1087.117,384.139,-97.557,177.311,25.990,154.210
C08657=1087.111,383.918,-97.523,177.309,25.984,154.209
C08658=1087.106,383.697,-97.489,177.306,25.977,154.208
C08659=1087.101,383.476,-97.455,177.303,25.972,154.207
C08660=1087.095,383.229,-97.417,177.300,25.965,154.205
C08661=1087.088,382.982,-97.379,177.296,25.958,154.204
C08662=1087.082,382.735,-97.341,177.293,25.951,154.203
C08663=1087.077,382.488,-97.303,177.290,25.944,154.202
C08664=1087.070,382.241,-97.266,177.286,25.938,154.200
C08665=1087.064,381.994,-97.228,177.283,25.931,154.199
C08666=1087.058,381.747,-97.191,177.280,25.925,154.198
C08667=1087.052,381.499,-97.153,177.277,25.918,154.197
C08668=1087.046,381.253,-97.115,177.274,25.912,154.196
C08669=1087.040,381.006,-97.077,177.270,25.905,154.194
C08670=1087.033,380.759,-97.040,177.267,25.899,154.193
C08671=1087.027,380.511,-97.003,177.264,25.892,154.192
C08672=1087.021,380.265,-96.965,177.260,25.886,154.191
C08673=1087.016,380.018,-96.927,177.257,25.879,154.190
C08674=1087.008,379.771,-96.890,177.254,25.873,154.189
C08675=1087.003,379.523,-96.853,177.251,25.867,154.188
C08676=1086.997,379.277,-96.815,177.248,25.860,154.186
C08677=1086.991,379.030,-96.777,177.244,25.854,154.185
C08678=1086.984,378.782,-96.740,177.241,25.847,154.184
C08679=1086.978,378.535,-96.702,177.238,25.841,154.183
C08680=1086.972,378.288,-96.665,177.235,25.834,154.182
C08681=1086.967,378.041,-96.628,177.232,25.828,154.181
C08682=1086.960,377.795,-96.591,177.228,25.822,154.179
C08683=1086.954,377.548,-96.553,177.225,25.816,154.178
C08684=1086.948,377.300,-96.515,177.222,25.809,154.177
C08685=1086.941,377.053,-96.479,177.218,25.803,154.176
C08686=1086.936,376.806,-96.441,177.216,25.797,154.175
C08687=1086.930,376.559,-96.404,177.212,25.791,154.174
C08688=1086.924,376.312,-96.367,177.209,25.784,154.173
C08689=1086.918,376.065,-96.330,177.205,25.778,154.172
C08690=1086.912,375.818,-96.293,177.202,25.771,154.170
C08691=1086.906,375.571,-96.255,177.200,25.765,154.169
C08692=1086.900,375.324,-96.219,177.196,25.759,154.168
C08693=1086.894,375.076,-96.181,177.193,25.753,154.167
C08694=1086.888,374.829,-96.144,177.189,25.747,154.166
C08695=1086.881,374.582,-96.107,177.187,25.741,154.165
C08696=1086.876,374.335,-96.070,177.184,25.734,154.164
C08697=1086.869,374.088,-96.034,177.180,25.728,154.163
C08698=1086.864,373.841,-95.996,177.177,25.722,154.162
C08699=1086.857,373.594,-95.959,177.174,25.716,154.161
C08700=1086.852,373.347,-95.922,177.171,25.710,154.160
C08701=1086.845,373.100,-95.886,177.167,25.704,154.159
C08702=1086.840,372.852,-95.849,177.164,25.698,154.158
C08703=1086.833,372.606,-95.812,177.161,25.692,154.156
C08704=1086.827,372.359,-95.775,177.158,25.686,154.155
C08705=1086.821,372.111,-95.738,177.154,25.680,154.154
C08706=1086.815,371.864,-95.702,177.151,25.674,154.153
C08707=1086.809,371.617,-95.665,177.148,25.668,154.152
C08708=1086.799,371.202,-95.603,177.143,25.658,154.151
C08709=1086.789,370.787,-95.541,177.137,25.648,154.149
C08710=1086.778,370.373,-95.480,177.132,25.638,154.147
C08711=1086.768,369.958,-95.418,177.127,25.628,154.145
C08712=1086.760,369.605,-95.367,177.122,25.620,154.144
C08713=1086.751,369.253,-95.314,177.118,25.612,154.143
C08714=1086.742,368.899,-95.262,177.113,25.603,154.141
C08715=1086.734,368.547,-95.210,177.108,25.595,154.140
C08716=1086.727,368.300,-95.174,177.105,25.589,154.139
C08717=1086.721,368.052,-95.138,177.102,25.583,154.138
C08718=1086.716,367.805,-95.101,177.099,25.577,154.137
C08719=1086.710,367.558,-95.065,177.096,25.572,154.136
C08720=1086.704,367.311,-95.028,177.092,25.566,154.135
C08721=1086.698,367.064,-94.993,177.089,25.560,154.134
C08722=1086.692,366.816,-94.956,177.086,25.555,154.133
C08723=1086.686,366.569,-94.919,177.083,25.548,154.132
C08724=1086.680,366.322,-94.883,177.080,25.543,154.131
C08725=1086.674,366.074,-94.846,177.077,25.537,154.130
C08726=1086.669,365.827,-94.811,177.073,25.531,154.129
C08727=1086.662,365.580,-94.775,177.070,25.525,154.128
C08728=1086.656,365.333,-94.738,177.067,25.520,154.127
C08729=1086.650,365.085,-94.702,177.064,25.514,154.126
C08730=1086.644,364.838,-94.666,177.060,25.509,154.125
C08731=1086.638,364.591,-94.630,177.058,25.503,154.124
C08732=1086.632,364.343,-94.593,177.054,25.498,154.123
C08733=1086.627,364.096,-94.558,177.052,25.492,154.122
C08734=1086.620,363.849,-94.521,177.048,25.487,154.121
C08735=1086.614,363.602,-94.486,177.044,25.481,154.120
C08736=1086.608,363.354,-94.450,177.042,25.476,154.119
C08737=1086.602,363.107,-94.413,177.038,25.470,154.119
C08738=1086.596,362.859,-94.378,177.035,25.464,154.118
C08739=1086.590,362.613,-94.342,177.032,25.459,154.117
C08740=1086.584,362.365,-94.306,177.029,25.453,154.116
C08741=1086.578,362.118,-94.270,177.026,25.448,154.115
C08742=1086.572,361.870,-94.235,177.023,25.442,154.114
C08743=1086.566,361.624,-94.198,177.019,25.437,154.113
C08744=1086.560,361.376,-94.163,177.016,25.432,154.112
C08745=1086.554,361.128,-94.127,177.013,25.426,154.111
C08746=1086.548,360.880,-94.091,177.010,25.420,154.110
C08747=1086.542,360.634,-94.055,177.007,25.415,154.109
C08748=1086.536,360.386,-94.019,177.004,25.410,154.109
C08749=1086.530,360.139,-93.984,177.000,25.404,154.108
C08750=1086.524,359.891,-93.949,176.997,25.398,154.107
C08751=1086.518,359.644,-93.913,176.994,25.394,154.106
C08752=1086.512,359.397,-93.877,176.991,25.388,154.105
C08753=1086.506,359.149,-93.842,176.988,25.383,154.104
C08754=1086.500,358.903,-93.806,176.984,25.377,154.103
C08755=1086.494,358.655,-93.770,176.982,25.372,154.102
C08756=1086.488,358.408,-93.735,176.978,25.367,154.101
C08757=1086.482,358.161,-93.699,176.976,25.362,154.101
C08758=1086.476,357.913,-93.664,176.972,25.356,154.100
C08759=1086.470,357.665,-93.628,176.968,25.351,154.099
C08760=1086.463,357.372,-93.586,176.965,25.345,154.098
C08761=1086.455,357.079,-93.545,176.962,25.338,154.097
C08762=1086.449,356.785,-93.502,176.957,25.332,154.096
C08763=1086.441,356.492,-93.461,176.954,25.326,154.095
C08764=1086.436,356.245,-93.425,176.950,25.320,154.094
C08765=1086.430,355.997,-93.390,176.948,25.316,154.093
C08766=1086.424,355.750,-93.355,176.944,25.310,154.092
C08767=1086.418,355.503,-93.319,176.941,25.305,154.092
C08768=1086.412,355.254,-93.284,176.938,25.300,154.091
C08769=1086.407,355.007,-93.249,176.935,25.295,154.090
C08770=1086.400,354.760,-93.214,176.932,25.290,154.089
C08771=1086.394,354.513,-93.178,176.929,25.285,154.088
C08772=1086.389,354.265,-93.143,176.925,25.279,154.087
C08773=1086.383,354.018,-93.108,176.923,25.274,154.087
C08774=1086.377,353.770,-93.073,176.919,25.269,154.086
C08775=1086.370,353.523,-93.037,176.916,25.264,154.085
C08776=1086.365,353.275,-93.003,176.913,25.259,154.084
C08777=1086.359,353.028,-92.967,176.910,25.254,154.083
C08778=1086.353,352.780,-92.932,176.906,25.248,154.083
C08779=1086.347,352.533,-92.897,176.904,25.244,154.082
C08780=1086.341,352.286,-92.862,176.900,25.238,154.081
C08781=1086.335,352.038,-92.828,176.897,25.233,154.080
C08782=1086.329,351.791,-92.792,176.895,25.229,154.079
C08783=1086.323,351.543,-92.758,176.891,25.223,154.078
C08784=1086.317,351.296,-92.722,176.888,25.218,154.078
C08785=1086.311,351.048,-92.688,176.885,25.213,154.077
C08786=1086.306,350.801,-92.653,176.882,25.208,154.076
C08787=1086.299,350.553,-92.618,176.878,25.203,154.075
C08788=1086.294,350.306,-92.583,176.876,25.199,154.075
C08789=1086.287,350.058,-92.548,176.872,25.193,154.074
C08790=1086.282,349.810,-92.514,176.869,25.188,154.073
C08791=1086.275,349.563,-92.479,176.866,25.183,154.072
C08792=1086.270,349.316,-92.445,176.863,25.178,154.071
C08793=1086.263,349.068,-92.409,176.860,25.174,154.071
C08794=1086.258,348.821,-92.375,176.857,25.169,154.070
C08795=1086.252,348.572,-92.340,176.854,25.164,154.069
C08796=1086.246,348.326,-92.305,176.850,25.159,154.068
C08797=1086.241,348.078,-92.270,176.847,25.154,154.068
C08798=1086.234,347.830,-92.236,176.845,25.149,154.067
C08799=1086.228,347.583,-92.202,176.841,25.144,154.066
C08800=1086.222,347.335,-92.166,176.838,25.139,154.065
C08801=1086.216,347.088,-92.132,176.835,25.134,154.065
C08802=1086.211,346.841,-92.098,176.832,25.130,154.064
C08803=1086.205,346.592,-92.063,176.828,25.124,154.063
C08804=1086.199,346.345,-92.029,176.825,25.120,154.062
C08805=1086.193,346.098,-91.995,176.823,25.115,154.062
C08806=1086.187,345.850,-91.959,176.819,25.110,154.061
C08807=1086.181,345.603,-91.925,176.816,25.105,154.060
C08808=1086.175,345.355,-91.891,176.813,25.100,154.059
C08809=1086.170,345.107,-91.856,176.810,25.096,154.059
C08810=1086.164,344.860,-91.822,176.807,25.091,154.058
C08811=1086.157,344.612,-91.788,176.804,25.086,154.057
C08812=1086.149,344.216,-91.733,176.799,25.078,154.056
C08813=1086.139,343.820,-91.678,176.794,25.071,154.055
C08814=1086.129,343.424,-91.623,176.789,25.063,154.054
C08815=1086.120,343.027,-91.568,176.784,25.056,154.053
C08816=1086.114,342.780,-91.534,176.781,25.051,154.052
C08817=1086.108,342.533,-91.500,176.778,25.047,154.051
C08818=1086.101,342.285,-91.466,176.774,25.042,154.051
C08819=1086.096,342.037,-91.432,176.772,25.037,154.050
C08820=1086.090,341.789,-91.398,176.769,25.032,154.049
C08821=1086.085,341.542,-91.364,176.765,25.028,154.048
C08822=1086.078,341.294,-91.329,176.762,25.023,154.048
C08823=1086.073,341.047,-91.295,176.760,25.019,154.047
C08824=1086.067,340.799,-91.261,176.756,25.014,154.046
C08825=1086.061,340.551,-91.228,176.753,25.009,154.046
C08826=1086.055,340.303,-91.193,176.750,25.004,154.045
C08827=1086.049,340.056,-91.159,176.747,25.000,154.044
C08828=1086.043,339.808,-91.126,176.744,24.995,154.044
C08829=1086.037,339.561,-91.092,176.741,24.991,154.043
C08830=1086.032,339.314,-91.058,176.737,24.986,154.042
C08831=1086.025,339.065,-91.024,176.735,24.982,154.042
C08832=1086.020,338.818,-90.990,176.732,24.977,154.041
C08833=1086.014,338.570,-90.956,176.728,24.972,154.040
C08834=1086.008,338.323,-90.923,176.725,24.968,154.040
C08835=1086.002,338.075,-90.889,176.722,24.963,154.039
C08836=1085.996,337.827,-90.855,176.720,24.959,154.038
C08837=1085.990,337.579,-90.821,176.716,24.954,154.038
C08838=1085.985,337.331,-90.788,176.713,24.950,154.037
C08839=1085.979,337.084,-90.754,176.710,24.945,154.036
C08840=1085.973,336.837,-90.720,176.707,24.940,154.036
C08841=1085.967,336.589,-90.687,176.704,24.936,154.035
C08842=1085.961,336.341,-90.653,176.701,24.932,154.034
C08843=1085.955,336.093,-90.619,176.697,24.927,154.034
C08844=1085.949,335.846,-90.586,176.694,24.923,154.033
C08845=1085.943,335.598,-90.552,176.692,24.918,154.032
C08846=1085.938,335.350,-90.518,176.689,24.914,154.032
C08847=1085.932,335.103,-90.484,176.685,24.909,154.031
C08848=1085.926,334.855,-90.452,176.682,24.905,154.030
C08849=1085.920,334.608,-90.418,176.679,24.901,154.030
C08850=1085.914,334.360,-90.384,176.677,24.896,154.029
C08851=1085.908,334.112,-90.350,176.673,24.891,154.028
C08852=1085.902,333.864,-90.317,176.670,24.887,154.028
C08853=1085.896,333.616,-90.284,176.667,24.883,154.027
C08854=1085.890,333.369,-90.250,176.664,24.878,154.026
C08855=1085.885,333.121,-90.217,176.661,24.874,154.026
C08856=1085.879,332.873,-90.184,176.658,24.870,154.025
C08857=1085.873,332.625,-90.151,176.655,24.865,154.025
C08858=1085.867,332.378,-90.117,176.652,24.861,154.024
C08859=1085.861,332.130,-90.084,176.648,24.856,154.023
C08860=1085.856,331.882,-90.050,176.646,24.852,154.023
C08861=1085.850,331.635,-90.017,176.643,24.847,154.022
C08862=1085.844,331.387,-89.984,176.640,24.843,154.021
C08863=1085.838,331.139,-89.951,176.637,24.839,154.021
C08864=1085.828,330.737,-89.897,176.632,24.832,154.020
C08865=1085.819,330.336,-89.843,176.627,24.825,154.019
C08866=1085.808,329.934,-89.790,176.622,24.818,154.018
C08867=1085.799,329.532,-89.736,176.617,24.812,154.017
C08868=1085.793,329.284,-89.704,176.614,24.807,154.016
C08869=1085.787,329.036,-89.670,176.611,24.803,154.016
C08870=1085.781,328.789,-89.638,176.608,24.799,154.015
C08871=1085.776,328.541,-89.604,176.604,24.794,154.015
C08872=1085.769,328.293,-89.571,176.601,24.790,154.014
C08873=1085.764,328.045,-89.538,176.598,24.786,154.014
C08874=1085.757,327.798,-89.505,176.596,24.782,154.013
C08875=1085.751,327.550,-89.473,176.593,24.778,154.012
C08876=1085.746,327.302,-89.440,176.589,24.774,154.012
C08877=1085.740,327.054,-89.407,176.586,24.769,154.011
C08878=1085.734,326.806,-89.374,176.583,24.765,154.011
C08879=1085.728,326.559,-89.341,176.580,24.761,154.010
C08880=1085.721,326.311,-89.308,176.577,24.757,154.010
C08881=1085.716,326.063,-89.275,176.575,24.753,154.009
C08882=1085.710,325.815,-89.243,176.571,24.748,154.008
C08883=1085.704,325.567,-89.210,176.568,24.744,154.008
C08884=1085.698,325.319,-89.177,176.565,24.740,154.007
C08885=1085.693,325.072,-89.145,176.562,24.736,154.007
C08886=1085.687,324.824,-89.112,176.559,24.732,154.006
C08887=1085.681,324.576,-89.079,176.556,24.728,154.005
C08888=1085.675,324.329,-89.047,176.554,24.724,154.005
C08889=1085.669,324.080,-89.014,176.550,24.719,154.004
C08890=1085.663,323.833,-88.981,176.547,24.715,154.004
C08891=1085.657,323.584,-88.949,176.544,24.711,154.003
C08892=1085.652,323.337,-88.916,176.541,24.707,154.003
C08893=1085.646,323.090,-88.883,176.538,24.703,154.002
C08894=1085.640,322.841,-88.851,176.535,24.699,154.002
C08895=1085.634,322.594,-88.818,176.532,24.695,154.001
C08896=1085.628,322.345,-88.786,176.529,24.690,154.000
C08897=1085.623,322.098,-88.754,176.526,24.686,154.000
C08898=1085.617,321.850,-88.721,176.523,24.682,153.999
C08899=1085.611,321.602,-88.688,176.520,24.678,153.999
C08900=1085.605,321.354,-88.656,176.517,24.674,153.998
C08901=1085.599,321.107,-88.624,176.514,24.670,153.998
C08902=1085.594,320.859,-88.591,176.511,24.666,153.997
C08903=1085.588,320.611,-88.559,176.508,24.662,153.997
C08904=1085.582,320.363,-88.526,176.506,24.658,153.996
C08905=1085.576,320.116,-88.494,176.502,24.654,153.995
C08906=1085.571,319.867,-88.461,176.499,24.649,153.995
C08907=1085.565,319.619,-88.429,176.496,24.645,153.994
C08908=1085.559,319.372,-88.397,176.493,24.641,153.994
C08909=1085.553,319.124,-88.365,176.490,24.637,153.993
C08910=1085.548,318.876,-88.332,176.487,24.633,153.993
C08911=1085.542,318.629,-88.300,176.484,24.629,153.992
C08912=1085.536,318.380,-88.268,176.482,24.625,153.992
C08913=1085.530,318.132,-88.236,176.479,24.621,153.991
C08914=1085.525,317.885,-88.204,176.476,24.617,153.990
C08915=1085.519,317.637,-88.171,176.473,24.613,153.990
C08916=1085.510,317.228,-88.119,176.468,24.607,153.989
C08917=1085.500,316.820,-88.065,176.463,24.600,153.988
C08918=1085.491,316.411,-88.012,176.458,24.593,153.987
C08919=1085.482,316.003,-87.960,176.453,24.587,153.986
C08920=1085.476,315.754,-87.928,176.450,24.583,153.986
C08921=1085.471,315.507,-87.896,176.447,24.579,153.985
C08922=1085.465,315.258,-87.864,176.444,24.574,153.985
C08923=1085.459,315.011,-87.831,176.441,24.570,153.984
C08924=1085.454,314.763,-87.799,176.438,24.567,153.984
C08925=1085.447,314.515,-87.768,176.435,24.563,153.983
C08926=1085.441,314.267,-87.736,176.432,24.559,153.983
C08927=1085.436,314.020,-87.704,176.429,24.555,153.982
C08928=1085.430,313.771,-87.672,176.426,24.551,153.982
C08929=1085.424,313.523,-87.640,176.423,24.548,153.981
C08930=1085.418,313.276,-87.609,176.420,24.544,153.981
C08931=1085.412,313.028,-87.577,176.417,24.540,153.980
C08932=1085.406,312.780,-87.545,176.414,24.536,153.980
C08933=1085.400,312.531,-87.514,176.411,24.532,153.979
C08934=1085.394,312.283,-87.483,176.408,24.528,153.979
C08935=1085.388,312.036,-87.451,176.405,24.524,153.978
C08936=1085.382,311.788,-87.419,176.403,24.520,153.978
C08937=1085.376,311.541,-87.388,176.400,24.517,153.977
C08938=1085.370,311.292,-87.356,176.397,24.513,153.977
C08939=1085.365,311.045,-87.324,176.394,24.509,153.976
C08940=1085.359,310.797,-87.292,176.391,24.505,153.976
C08941=1085.352,310.548,-87.261,176.388,24.502,153.975
C08942=1085.347,310.301,-87.230,176.385,24.498,153.975
C08943=1085.341,310.052,-87.198,176.382,24.494,153.974
C08944=1085.335,309.805,-87.167,176.379,24.490,153.974
C08945=1085.329,309.557,-87.135,176.376,24.487,153.974
C08946=1085.324,309.309,-87.104,176.373,24.483,153.973
C08947=1085.318,309.062,-87.073,176.370,24.479,153.972
C08948=1085.312,308.813,-87.040,176.366,24.475,153.972
C08949=1085.307,308.565,-87.010,176.363,24.471,153.972
C08950=1085.300,308.317,-86.978,176.360,24.467,153.971
C08951=1085.295,308.070,-86.946,176.357,24.463,153.971
C08952=1085.289,307.821,-86.915,176.354,24.460,153.970
C08953=1085.283,307.574,-86.884,176.352,24.456,153.970
C08954=1085.277,307.326,-86.852,176.348,24.452,153.969
C08955=1085.272,307.077,-86.821,176.346,24.448,153.969
C08956=1085.266,306.830,-86.790,176.343,24.444,153.968
C08957=1085.260,306.581,-86.759,176.340,24.441,153.968
C08958=1085.254,306.334,-86.728,176.337,24.437,153.967
C08959=1085.248,306.086,-86.696,176.334,24.433,153.967
C08960=1085.243,305.838,-86.665,176.331,24.429,153.966
C08961=1085.237,305.591,-86.634,176.328,24.426,153.966
C08962=1085.231,305.342,-86.602,176.325,24.422,153.965
C08963=1085.225,305.095,-86.571,176.322,24.418,153.965
C08964=1085.220,304.846,-86.540,176.319,24.414,153.964
C08965=1085.213,304.599,-86.509,176.316,24.411,153.964
C08966=1085.208,304.350,-86.478,176.314,24.407,153.963
C08967=1085.203,304.102,-86.447,176.311,24.403,153.963
C08968=1085.193,303.697,-86.396,176.306,24.397,153.962
C08969=1085.183,303.292,-86.345,176.301,24.391,153.962
C08970=1085.175,302.885,-86.295,176.296,24.385,153.961
C08971=1085.165,302.480,-86.244,176.292,24.379,153.960
C08972=1085.159,302.231,-86.213,176.289,24.375,153.960
C08973=1085.153,301.983,-86.182,176.286,24.371,153.959
C08974=1085.148,301.736,-86.151,176.283,24.368,153.959
C08975=1085.142,301.488,-86.120,176.280,24.364,153.958
C08976=1085.137,301.240,-86.089,176.277,24.360,153.958
C08977=1085.131,300.991,-86.058,176.274,24.357,153.957
C08978=1085.125,300.744,-86.027,176.271,24.353,153.957
C08979=1085.119,300.496,-85.996,176.268,24.349,153.956
C08980=1085.114,300.248,-85.966,176.265,24.346,153.956
C08981=1085.109,300.000,-85.935,176.262,24.342,153.955
C08982=1085.103,299.751,-85.904,176.259,24.338,153.955
C08983=1085.097,299.504,-85.873,176.256,24.334,153.954
C08984=1085.092,299.256,-85.842,176.253,24.330,153.954
C08985=1085.086,299.008,-85.812,176.250,24.327,153.954
C08986=1085.080,298.760,-85.781,176.248,24.323,153.953
C08987=1085.075,298.512,-85.750,176.245,24.319,153.953
C08988=1085.069,298.264,-85.720,176.242,24.316,153.952
C08989=1085.063,298.015,-85.689,176.240,24.312,153.952
C08990=1085.058,297.768,-85.658,176.237,24.308,153.951
C08991=1085.052,297.520,-85.628,176.234,24.305,153.951
C08992=1085.046,297.272,-85.598,176.231,24.301,153.950
C08993=1085.041,297.024,-85.567,176.228,24.297,153.950
C08994=1085.035,296.775,-85.536,176.225,24.294,153.950
C08995=1085.029,296.527,-85.505,176.222,24.290,153.949
C08996=1085.023,296.280,-85.475,176.219,24.287,153.949
C08997=1085.018,296.032,-85.444,176.216,24.283,153.948
C08998=1085.012,295.784,-85.414,176.213,24.280,153.948
C08999=1085.006,295.536,-85.383,176.210,24.276,153.948
C09000=1085.000,295.287,-85.353,176.208,24.272,153.947
C09001=1084.994,295.040,-85.322,176.205,24.269,153.947
C09002=1084.988,294.791,-85.293,176.202,24.265,153.946
C09003=1084.983,294.543,-85.262,176.199,24.262,153.946
C09004=1084.977,294.295,-85.232,176.196,24.258,153.945
C09005=1084.971,294.048,-85.202,176.193,24.255,153.945
C09006=1084.966,293.799,-85.171,176.190,24.251,153.945
C09007=1084.960,293.552,-85.140,176.187,24.247,153.944
C09008=1084.954,293.303,-85.110,176.184,24.244,153.944
C09009=1084.948,293.055,-85.080,176.182,24.241,153.943
C09010=1084.942,292.807,-85.050,176.179,24.237,153.943
C09011=1084.936,292.559,-85.019,176.176,24.234,153.942
C09012=1084.931,292.311,-84.990,176.173,24.230,153.942
C09013=1084.925,292.063,-84.959,176.170,24.226,153.942
C09014=1084.919,291.815,-84.929,176.167,24.222,153.941
C09015=1084.914,291.567,-84.899,176.164,24.219,153.941
C09016=1084.908,291.319,-84.869,176.161,24.215,153.940
C09017=1084.902,291.071,-84.839,176.159,24.212,153.940
C09018=1084.897,290.822,-84.809,176.156,24.209,153.939
C09019=1084.891,290.575,-84.779,176.153,24.205,153.939
C09020=1084.881,290.183,-84.731,176.148,24.200,153.938
C09021=1084.873,289.792,-84.684,176.144,24.194,153.938
C09022=1084.864,289.399,-84.636,176.139,24.188,153.937
C09023=1084.855,289.008,-84.590,176.135,24.183,153.936
C09024=1084.849,288.760,-84.560,176.132,24.180,153.936
C09025=1084.843,288.511,-84.530,176.129,24.176,153.936
C09026=1084.837,288.263,-84.499,176.126,24.172,153.935
C09027=1084.831,288.015,-84.470,176.123,24.169,153.935
C09028=1084.825,287.767,-84.439,176.120,24.166,153.935
C09029=1084.819,287.519,-84.410,176.117,24.162,153.934
C09030=1084.813,287.271,-84.380,176.115,24.159,153.934
C09031=1084.808,287.022,-84.350,176.112,24.155,153.933
C09032=1084.803,286.775,-84.321,176.109,24.152,153.933
C09033=1084.797,286.527,-84.291,176.106,24.148,153.933
C09034=1084.791,286.279,-84.262,176.103,24.145,153.932
C09035=1084.785,286.030,-84.232,176.100,24.141,153.932
C09036=1084.780,285.783,-84.202,176.097,24.138,153.931
C09037=1084.774,285.534,-84.172,176.094,24.135,153.931
C09038=1084.769,285.286,-84.143,176.092,24.131,153.931
C09039=1084.762,285.038,-84.113,176.089,24.128,153.930
C09040=1084.757,284.790,-84.083,176.086,24.124,153.930
C09041=1084.751,284.541,-84.054,176.083,24.121,153.929
C09042=1084.745,284.293,-84.024,176.080,24.117,153.929
C09043=1084.739,284.045,-83.994,176.077,24.114,153.929
C09044=1084.733,283.797,-83.964,176.074,24.110,153.928
C09045=1084.728,283.548,-83.935,176.071,24.107,153.928
C09046=1084.723,283.301,-83.906,176.068,24.104,153.928
C09047=1084.717,283.053,-83.877,176.066,24.100,153.927
C09048=1084.711,282.804,-83.847,176.063,24.097,153.927
C09049=1084.705,282.556,-83.817,176.060,24.093,153.926
C09050=1084.699,282.308,-83.788,176.057,24.090,153.926
C09051=1084.694,282.060,-83.758,176.054,24.086,153.925
C09052=1084.689,281.812,-83.729,176.052,24.083,153.925
C09053=1084.682,281.564,-83.700,176.049,24.080,153.925
C09054=1084.677,281.315,-83.670,176.046,24.076,153.924
C09055=1084.671,281.067,-83.640,176.043,24.073,153.924
C09056=1084.665,280.819,-83.611,176.041,24.069,153.924
C09057=1084.660,280.570,-83.582,176.038,24.066,153.923
C09058=1084.653,280.322,-83.553,176.035,24.063,153.923
C09059=1084.649,280.075,-83.523,176.032,24.059,153.922
C09060=1084.643,279.826,-83.494,176.029,24.056,153.922
C09061=1084.637,279.578,-83.465,176.027,24.052,153.922
C09062=1084.631,279.329,-83.435,176.024,24.049,153.921
C09063=1084.625,279.081,-83.406,176.021,24.046,153.921
C09064=1084.620,278.834,-83.377,176.018,24.042,153.921
C09065=1084.614,278.585,-83.348,176.016,24.039,153.920
C09066=1084.609,278.336,-83.319,176.013,24.036,153.920
C09067=1084.602,278.088,-83.290,176.010,24.032,153.919
C09068=1084.597,277.840,-83.260,176.007,24.029,153.919
C09069=1084.591,277.592,-83.231,176.004,24.025,153.919
C09070=1084.586,277.344,-83.202,176.001,24.022,153.918
C09071=1084.580,277.096,-83.173,175.998,24.019,153.918
C09072=1084.571,276.714,-83.128,175.994,24.013,153.917
C09073=1084.562,276.332,-83.084,175.989,24.009,153.917
C09074=1084.553,275.950,-83.039,175.986,24.004,153.916
C09075=1084.545,275.567,-82.995,175.981,23.998,153.916
C09076=1084.539,275.319,-82.965,175.978,23.995,153.915
C09077=1084.533,275.071,-82.936,175.975,23.992,153.915
C09078=1084.527,274.823,-82.907,175.973,23.988,153.915
C09079=1084.522,274.575,-82.879,175.970,23.985,153.914
C09080=1084.516,274.326,-82.849,175.967,23.982,153.914
C09081=1084.511,274.078,-82.821,175.964,23.978,153.913
C09082=1084.504,273.830,-82.792,175.962,23.975,153.913
C09083=1084.499,273.582,-82.763,175.959,23.972,153.913
C09084=1084.494,273.333,-82.735,175.956,23.968,153.912
C09085=1084.487,273.085,-82.706,175.953,23.965,153.912
C09086=1084.482,272.836,-82.677,175.951,23.962,153.912
C09087=1084.476,272.588,-82.648,175.948,23.958,153.911
C09088=1084.470,272.341,-82.619,175.945,23.955,153.911
C09089=1084.464,272.092,-82.591,175.943,23.952,153.911
C09090=1084.459,271.844,-82.561,175.940,23.948,153.910
C09091=1084.453,271.595,-82.533,175.936,23.945,153.910
